   // GBK_TO_UNICODE[9557] := 16#6B54;
   // GBK_TO_UNICODE[9558] := 16#9A5C;
   // GBK_TO_UNICODE[9559] := 16#6B55;
   // GBK_TO_UNICODE[9560] := 16#9A5D;
   // GBK_TO_UNICODE[9561] := 16#6B56;
   // GBK_TO_UNICODE[9562] := 16#9A5E;
   // GBK_TO_UNICODE[9563] := 16#6B57;
   // GBK_TO_UNICODE[9564] := 16#9A5F;
   // GBK_TO_UNICODE[9565] := 16#6B58;
   // GBK_TO_UNICODE[9566] := 16#9A60;
   // GBK_TO_UNICODE[9567] := 16#6B5A;
   // GBK_TO_UNICODE[9568] := 16#9A61;
   // GBK_TO_UNICODE[9569] := 16#6B5B;
   // GBK_TO_UNICODE[9570] := 16#9A62;
   // GBK_TO_UNICODE[9571] := 16#6B5C;
   // GBK_TO_UNICODE[9572] := 16#9A63;
   // GBK_TO_UNICODE[9573] := 16#6B5D;
   // GBK_TO_UNICODE[9574] := 16#9A64;
   // GBK_TO_UNICODE[9575] := 16#6B5E;
   // GBK_TO_UNICODE[9576] := 16#9A65;
   // GBK_TO_UNICODE[9577] := 16#6B5F;
   // GBK_TO_UNICODE[9578] := 16#9A66;
   // GBK_TO_UNICODE[9579] := 16#6B60;
   // GBK_TO_UNICODE[9580] := 16#9A67;
   // GBK_TO_UNICODE[9581] := 16#6B61;
   // GBK_TO_UNICODE[9582] := 16#9A68;
   // GBK_TO_UNICODE[9583] := 16#6B68;
   // GBK_TO_UNICODE[9584] := 16#9A69;
   // GBK_TO_UNICODE[9585] := 16#6B69;
   // GBK_TO_UNICODE[9586] := 16#9A6A;
   // GBK_TO_UNICODE[9587] := 16#6B6B;
   // GBK_TO_UNICODE[9588] := 16#9A6B;
   // GBK_TO_UNICODE[9589] := 16#6B6C;
   // GBK_TO_UNICODE[9590] := 16#9A6C;
   // GBK_TO_UNICODE[9591] := 16#6B6D;
   // GBK_TO_UNICODE[9592] := 16#9A6D;
   // GBK_TO_UNICODE[9593] := 16#6B6E;
   // GBK_TO_UNICODE[9594] := 16#9A6E;
   // GBK_TO_UNICODE[9595] := 16#6B6F;
   // GBK_TO_UNICODE[9596] := 16#9A6F;
   // GBK_TO_UNICODE[9597] := 16#6B70;
   // GBK_TO_UNICODE[9598] := 16#9A70;
   // GBK_TO_UNICODE[9599] := 16#6B71;
   // GBK_TO_UNICODE[9600] := 16#9A71;
   // GBK_TO_UNICODE[9601] := 16#6B72;
   // GBK_TO_UNICODE[9602] := 16#9A72;
   // GBK_TO_UNICODE[9603] := 16#6B73;
   // GBK_TO_UNICODE[9604] := 16#9A73;
   // GBK_TO_UNICODE[9605] := 16#6B74;
   // GBK_TO_UNICODE[9606] := 16#9A74;
   // GBK_TO_UNICODE[9607] := 16#6B75;
   // GBK_TO_UNICODE[9608] := 16#9A75;
   // GBK_TO_UNICODE[9609] := 16#6B76;
   // GBK_TO_UNICODE[9610] := 16#9A76;
   // GBK_TO_UNICODE[9611] := 16#6B77;
   // GBK_TO_UNICODE[9612] := 16#9A77;
   // GBK_TO_UNICODE[9613] := 16#6B78;
   // GBK_TO_UNICODE[9614] := 16#9A78;
   // GBK_TO_UNICODE[9615] := 16#6B7A;
   // GBK_TO_UNICODE[9616] := 16#9A79;
   // GBK_TO_UNICODE[9617] := 16#6B7D;
   // GBK_TO_UNICODE[9618] := 16#9A7A;
   // GBK_TO_UNICODE[9619] := 16#6B7E;
   // GBK_TO_UNICODE[9620] := 16#9A7B;
   // GBK_TO_UNICODE[9621] := 16#6B7F;
   // GBK_TO_UNICODE[9622] := 16#9A7C;
   // GBK_TO_UNICODE[9623] := 16#6B80;
   // GBK_TO_UNICODE[9624] := 16#9A7D;
   // GBK_TO_UNICODE[9625] := 16#6B85;
   // GBK_TO_UNICODE[9626] := 16#9A7E;
   // GBK_TO_UNICODE[9627] := 16#6B88;
   // GBK_TO_UNICODE[9628] := 16#9A80;
   // GBK_TO_UNICODE[9629] := 16#6B8C;
   // GBK_TO_UNICODE[9630] := 16#9A81;
   // GBK_TO_UNICODE[9631] := 16#6B8E;
   // GBK_TO_UNICODE[9632] := 16#9A82;
   // GBK_TO_UNICODE[9633] := 16#6B8F;
   // GBK_TO_UNICODE[9634] := 16#9A83;
   // GBK_TO_UNICODE[9635] := 16#6B90;
   // GBK_TO_UNICODE[9636] := 16#9A84;
   // GBK_TO_UNICODE[9637] := 16#6B91;
   // GBK_TO_UNICODE[9638] := 16#9A85;
   // GBK_TO_UNICODE[9639] := 16#6B94;
   // GBK_TO_UNICODE[9640] := 16#9A86;
   // GBK_TO_UNICODE[9641] := 16#6B95;
   // GBK_TO_UNICODE[9642] := 16#9A87;
   // GBK_TO_UNICODE[9643] := 16#6B97;
   // GBK_TO_UNICODE[9644] := 16#9A88;
   // GBK_TO_UNICODE[9645] := 16#6B98;
   // GBK_TO_UNICODE[9646] := 16#9A89;
   // GBK_TO_UNICODE[9647] := 16#6B99;
   // GBK_TO_UNICODE[9648] := 16#9A8A;
   // GBK_TO_UNICODE[9649] := 16#6B9C;
   // GBK_TO_UNICODE[9650] := 16#9A8B;
   // GBK_TO_UNICODE[9651] := 16#6B9D;
   // GBK_TO_UNICODE[9652] := 16#9A8C;
   // GBK_TO_UNICODE[9653] := 16#6B9E;
   // GBK_TO_UNICODE[9654] := 16#9A8D;
   // GBK_TO_UNICODE[9655] := 16#6B9F;
   // GBK_TO_UNICODE[9656] := 16#9A8E;
   // GBK_TO_UNICODE[9657] := 16#6BA0;
   // GBK_TO_UNICODE[9658] := 16#9A8F;
   // GBK_TO_UNICODE[9659] := 16#6BA2;
   // GBK_TO_UNICODE[9660] := 16#9A90;
   // GBK_TO_UNICODE[9661] := 16#6BA3;
   // GBK_TO_UNICODE[9662] := 16#9A91;
   // GBK_TO_UNICODE[9663] := 16#6BA4;
   // GBK_TO_UNICODE[9664] := 16#9A92;
   // GBK_TO_UNICODE[9665] := 16#6BA5;
   // GBK_TO_UNICODE[9666] := 16#9A93;
   // GBK_TO_UNICODE[9667] := 16#6BA6;
   // GBK_TO_UNICODE[9668] := 16#9A94;
   // GBK_TO_UNICODE[9669] := 16#6BA7;
   // GBK_TO_UNICODE[9670] := 16#9A95;
   // GBK_TO_UNICODE[9671] := 16#6BA8;
   // GBK_TO_UNICODE[9672] := 16#9A96;
   // GBK_TO_UNICODE[9673] := 16#6BA9;
   // GBK_TO_UNICODE[9674] := 16#9A97;
   // GBK_TO_UNICODE[9675] := 16#6BAB;
   // GBK_TO_UNICODE[9676] := 16#9A98;
   // GBK_TO_UNICODE[9677] := 16#6BAC;
   // GBK_TO_UNICODE[9678] := 16#9A99;
   // GBK_TO_UNICODE[9679] := 16#6BAD;
   // GBK_TO_UNICODE[9680] := 16#9A9A;
   // GBK_TO_UNICODE[9681] := 16#6BAE;
   // GBK_TO_UNICODE[9682] := 16#9A9B;
   // GBK_TO_UNICODE[9683] := 16#6BAF;
   // GBK_TO_UNICODE[9684] := 16#9A9C;
   // GBK_TO_UNICODE[9685] := 16#6BB0;
   // GBK_TO_UNICODE[9686] := 16#9A9D;
   // GBK_TO_UNICODE[9687] := 16#6BB1;
   // GBK_TO_UNICODE[9688] := 16#9A9E;
   // GBK_TO_UNICODE[9689] := 16#6BB2;
   // GBK_TO_UNICODE[9690] := 16#9A9F;
   // GBK_TO_UNICODE[9691] := 16#6BB6;
   // GBK_TO_UNICODE[9692] := 16#9AA0;
   // GBK_TO_UNICODE[9693] := 16#6BB8;
   // GBK_TO_UNICODE[9694] := 16#9AA1;
   // GBK_TO_UNICODE[9695] := 16#6BB9;
   // GBK_TO_UNICODE[9696] := 16#9AA2;
   // GBK_TO_UNICODE[9697] := 16#6BBA;
   // GBK_TO_UNICODE[9698] := 16#9AA3;
   // GBK_TO_UNICODE[9699] := 16#6BBB;
   // GBK_TO_UNICODE[9700] := 16#9AA4;
   // GBK_TO_UNICODE[9701] := 16#6BBC;
   // GBK_TO_UNICODE[9702] := 16#9AA5;
   // GBK_TO_UNICODE[9703] := 16#6BBD;
   // GBK_TO_UNICODE[9704] := 16#9AA6;
   // GBK_TO_UNICODE[9705] := 16#6BBE;
   // GBK_TO_UNICODE[9706] := 16#9AA7;
   // GBK_TO_UNICODE[9707] := 16#6BC0;
   // GBK_TO_UNICODE[9708] := 16#9AA8;
   // GBK_TO_UNICODE[9709] := 16#6BC3;
   // GBK_TO_UNICODE[9710] := 16#9AA9;
   // GBK_TO_UNICODE[9711] := 16#6BC4;
   // GBK_TO_UNICODE[9712] := 16#9AAA;
   // GBK_TO_UNICODE[9713] := 16#6BC6;
   // GBK_TO_UNICODE[9714] := 16#9AAB;
   // GBK_TO_UNICODE[9715] := 16#6BC7;
   // GBK_TO_UNICODE[9716] := 16#9AAC;
   // GBK_TO_UNICODE[9717] := 16#6BC8;
   // GBK_TO_UNICODE[9718] := 16#9AAD;
   // GBK_TO_UNICODE[9719] := 16#6BC9;
   // GBK_TO_UNICODE[9720] := 16#9AAE;
   // GBK_TO_UNICODE[9721] := 16#6BCA;
   // GBK_TO_UNICODE[9722] := 16#9AAF;
   // GBK_TO_UNICODE[9723] := 16#6BCC;
   // GBK_TO_UNICODE[9724] := 16#9AB0;
   // GBK_TO_UNICODE[9725] := 16#6BCE;
   // GBK_TO_UNICODE[9726] := 16#9AB1;
   // GBK_TO_UNICODE[9727] := 16#6BD0;
   // GBK_TO_UNICODE[9728] := 16#9AB2;
   // GBK_TO_UNICODE[9729] := 16#6BD1;
   // GBK_TO_UNICODE[9730] := 16#9AB3;
   // GBK_TO_UNICODE[9731] := 16#6BD8;
   // GBK_TO_UNICODE[9732] := 16#9AB4;
   // GBK_TO_UNICODE[9733] := 16#6BDA;
   // GBK_TO_UNICODE[9734] := 16#9AB5;
   // GBK_TO_UNICODE[9735] := 16#6BDC;
   // GBK_TO_UNICODE[9736] := 16#9AB6;
   // GBK_TO_UNICODE[9737] := 16#6BDD;
   // GBK_TO_UNICODE[9738] := 16#9AB7;
   // GBK_TO_UNICODE[9739] := 16#6BDE;
   // GBK_TO_UNICODE[9740] := 16#9AB8;
   // GBK_TO_UNICODE[9741] := 16#6BDF;
   // GBK_TO_UNICODE[9742] := 16#9AB9;
   // GBK_TO_UNICODE[9743] := 16#6BE0;
   // GBK_TO_UNICODE[9744] := 16#9ABA;
   // GBK_TO_UNICODE[9745] := 16#6BE2;
   // GBK_TO_UNICODE[9746] := 16#9ABB;
   // GBK_TO_UNICODE[9747] := 16#6BE3;
   // GBK_TO_UNICODE[9748] := 16#9ABC;
   // GBK_TO_UNICODE[9749] := 16#6BE4;
   // GBK_TO_UNICODE[9750] := 16#9ABD;
   // GBK_TO_UNICODE[9751] := 16#6BE5;
   // GBK_TO_UNICODE[9752] := 16#9ABE;
   // GBK_TO_UNICODE[9753] := 16#6BE6;
   // GBK_TO_UNICODE[9754] := 16#9ABF;
   // GBK_TO_UNICODE[9755] := 16#6BE7;
   // GBK_TO_UNICODE[9756] := 16#9AC0;
   // GBK_TO_UNICODE[9757] := 16#6BE8;
   // GBK_TO_UNICODE[9758] := 16#9AC1;
   // GBK_TO_UNICODE[9759] := 16#6BE9;
   // GBK_TO_UNICODE[9760] := 16#9AC2;
   // GBK_TO_UNICODE[9761] := 16#6BEC;
   // GBK_TO_UNICODE[9762] := 16#9AC3;
   // GBK_TO_UNICODE[9763] := 16#6BED;
   // GBK_TO_UNICODE[9764] := 16#9AC4;
   // GBK_TO_UNICODE[9765] := 16#6BEE;
   // GBK_TO_UNICODE[9766] := 16#9AC5;
   // GBK_TO_UNICODE[9767] := 16#6BF0;
   // GBK_TO_UNICODE[9768] := 16#9AC6;
   // GBK_TO_UNICODE[9769] := 16#6BF1;
   // GBK_TO_UNICODE[9770] := 16#9AC7;
   // GBK_TO_UNICODE[9771] := 16#6BF2;
   // GBK_TO_UNICODE[9772] := 16#9AC8;
   // GBK_TO_UNICODE[9773] := 16#6BF4;
   // GBK_TO_UNICODE[9774] := 16#9AC9;
   // GBK_TO_UNICODE[9775] := 16#6BF6;
   // GBK_TO_UNICODE[9776] := 16#9ACA;
   // GBK_TO_UNICODE[9777] := 16#6BF7;
   // GBK_TO_UNICODE[9778] := 16#9ACB;
   // GBK_TO_UNICODE[9779] := 16#6BF8;
   // GBK_TO_UNICODE[9780] := 16#9ACC;
   // GBK_TO_UNICODE[9781] := 16#6BFA;
   // GBK_TO_UNICODE[9782] := 16#9ACD;
   // GBK_TO_UNICODE[9783] := 16#6BFB;
   // GBK_TO_UNICODE[9784] := 16#9ACE;
   // GBK_TO_UNICODE[9785] := 16#6BFC;
   // GBK_TO_UNICODE[9786] := 16#9ACF;
   // GBK_TO_UNICODE[9787] := 16#6BFE;
   // GBK_TO_UNICODE[9788] := 16#9AD0;
   // GBK_TO_UNICODE[9789] := 16#6BFF;
   // GBK_TO_UNICODE[9790] := 16#9AD1;
   // GBK_TO_UNICODE[9791] := 16#6C00;
   // GBK_TO_UNICODE[9792] := 16#9AD2;
   // GBK_TO_UNICODE[9793] := 16#6C01;
   // GBK_TO_UNICODE[9794] := 16#9AD3;
   // GBK_TO_UNICODE[9795] := 16#6C02;
   // GBK_TO_UNICODE[9796] := 16#9AD4;
   // GBK_TO_UNICODE[9797] := 16#6C03;
   // GBK_TO_UNICODE[9798] := 16#9AD5;
   // GBK_TO_UNICODE[9799] := 16#6C04;
   // GBK_TO_UNICODE[9800] := 16#9AD6;
   // GBK_TO_UNICODE[9801] := 16#6C08;
   // GBK_TO_UNICODE[9802] := 16#9AD7;
   // GBK_TO_UNICODE[9803] := 16#6C09;
   // GBK_TO_UNICODE[9804] := 16#9AD8;
   // GBK_TO_UNICODE[9805] := 16#6C0A;
   // GBK_TO_UNICODE[9806] := 16#9AD9;
   // GBK_TO_UNICODE[9807] := 16#6C0B;
   // GBK_TO_UNICODE[9808] := 16#9ADA;
   // GBK_TO_UNICODE[9809] := 16#6C0C;
   // GBK_TO_UNICODE[9810] := 16#9ADB;
   // GBK_TO_UNICODE[9811] := 16#6C0E;
   // GBK_TO_UNICODE[9812] := 16#9ADC;
   // GBK_TO_UNICODE[9813] := 16#6C12;
   // GBK_TO_UNICODE[9814] := 16#9ADD;
   // GBK_TO_UNICODE[9815] := 16#6C17;
   // GBK_TO_UNICODE[9816] := 16#9ADE;
   // GBK_TO_UNICODE[9817] := 16#6C1C;
   // GBK_TO_UNICODE[9818] := 16#9ADF;
   // GBK_TO_UNICODE[9819] := 16#6C1D;
   // GBK_TO_UNICODE[9820] := 16#9AE0;
   // GBK_TO_UNICODE[9821] := 16#6C1E;
   // GBK_TO_UNICODE[9822] := 16#9AE1;
   // GBK_TO_UNICODE[9823] := 16#6C20;
   // GBK_TO_UNICODE[9824] := 16#9AE2;
   // GBK_TO_UNICODE[9825] := 16#6C23;
   // GBK_TO_UNICODE[9826] := 16#9AE3;
   // GBK_TO_UNICODE[9827] := 16#6C25;
   // GBK_TO_UNICODE[9828] := 16#9AE4;
   // GBK_TO_UNICODE[9829] := 16#6C2B;
   // GBK_TO_UNICODE[9830] := 16#9AE5;
   // GBK_TO_UNICODE[9831] := 16#6C2C;
   // GBK_TO_UNICODE[9832] := 16#9AE6;
   // GBK_TO_UNICODE[9833] := 16#6C2D;
   // GBK_TO_UNICODE[9834] := 16#9AE7;
   // GBK_TO_UNICODE[9835] := 16#6C31;
   // GBK_TO_UNICODE[9836] := 16#9AE8;
   // GBK_TO_UNICODE[9837] := 16#6C33;
   // GBK_TO_UNICODE[9838] := 16#9AE9;
   // GBK_TO_UNICODE[9839] := 16#6C36;
   // GBK_TO_UNICODE[9840] := 16#9AEA;
   // GBK_TO_UNICODE[9841] := 16#6C37;
   // GBK_TO_UNICODE[9842] := 16#9AEB;
   // GBK_TO_UNICODE[9843] := 16#6C39;
   // GBK_TO_UNICODE[9844] := 16#9AEC;
   // GBK_TO_UNICODE[9845] := 16#6C3A;
   // GBK_TO_UNICODE[9846] := 16#9AED;
   // GBK_TO_UNICODE[9847] := 16#6C3B;
   // GBK_TO_UNICODE[9848] := 16#9AEE;
   // GBK_TO_UNICODE[9849] := 16#6C3C;
   // GBK_TO_UNICODE[9850] := 16#9AEF;
   // GBK_TO_UNICODE[9851] := 16#6C3E;
   // GBK_TO_UNICODE[9852] := 16#9AF0;
   // GBK_TO_UNICODE[9853] := 16#6C3F;
   // GBK_TO_UNICODE[9854] := 16#9AF1;
   // GBK_TO_UNICODE[9855] := 16#6C43;
   // GBK_TO_UNICODE[9856] := 16#9AF2;
   // GBK_TO_UNICODE[9857] := 16#6C44;
   // GBK_TO_UNICODE[9858] := 16#9AF3;
   // GBK_TO_UNICODE[9859] := 16#6C45;
   // GBK_TO_UNICODE[9860] := 16#9AF4;
   // GBK_TO_UNICODE[9861] := 16#6C48;
   // GBK_TO_UNICODE[9862] := 16#9AF5;
   // GBK_TO_UNICODE[9863] := 16#6C4B;
   // GBK_TO_UNICODE[9864] := 16#9AF6;
   // GBK_TO_UNICODE[9865] := 16#6C4C;
   // GBK_TO_UNICODE[9866] := 16#9AF7;
   // GBK_TO_UNICODE[9867] := 16#6C4D;
   // GBK_TO_UNICODE[9868] := 16#9AF8;
   // GBK_TO_UNICODE[9869] := 16#6C4E;
   // GBK_TO_UNICODE[9870] := 16#9AF9;
   // GBK_TO_UNICODE[9871] := 16#6C4F;
   // GBK_TO_UNICODE[9872] := 16#9AFA;
   // GBK_TO_UNICODE[9873] := 16#6C51;
   // GBK_TO_UNICODE[9874] := 16#9AFB;
   // GBK_TO_UNICODE[9875] := 16#6C52;
   // GBK_TO_UNICODE[9876] := 16#9AFC;
   // GBK_TO_UNICODE[9877] := 16#6C53;
   // GBK_TO_UNICODE[9878] := 16#9AFD;
   // GBK_TO_UNICODE[9879] := 16#6C56;
   // GBK_TO_UNICODE[9880] := 16#9AFE;
   // GBK_TO_UNICODE[9881] := 16#6C58;
   // GBK_TO_UNICODE[9882] := 16#9B40;
   // GBK_TO_UNICODE[9883] := 16#6C59;
   // GBK_TO_UNICODE[9884] := 16#9B41;
   // GBK_TO_UNICODE[9885] := 16#6C5A;
   // GBK_TO_UNICODE[9886] := 16#9B42;
   // GBK_TO_UNICODE[9887] := 16#6C62;
   // GBK_TO_UNICODE[9888] := 16#9B43;
   // GBK_TO_UNICODE[9889] := 16#6C63;
   // GBK_TO_UNICODE[9890] := 16#9B44;
   // GBK_TO_UNICODE[9891] := 16#6C65;
   // GBK_TO_UNICODE[9892] := 16#9B45;
   // GBK_TO_UNICODE[9893] := 16#6C66;
   // GBK_TO_UNICODE[9894] := 16#9B46;
   // GBK_TO_UNICODE[9895] := 16#6C67;
   // GBK_TO_UNICODE[9896] := 16#9B47;
   // GBK_TO_UNICODE[9897] := 16#6C6B;
   // GBK_TO_UNICODE[9898] := 16#9B48;
   // GBK_TO_UNICODE[9899] := 16#6C6C;
   // GBK_TO_UNICODE[9900] := 16#9B49;
   // GBK_TO_UNICODE[9901] := 16#6C6D;
   // GBK_TO_UNICODE[9902] := 16#9B4A;
   // GBK_TO_UNICODE[9903] := 16#6C6E;
   // GBK_TO_UNICODE[9904] := 16#9B4B;
   // GBK_TO_UNICODE[9905] := 16#6C6F;
   // GBK_TO_UNICODE[9906] := 16#9B4C;
   // GBK_TO_UNICODE[9907] := 16#6C71;
   // GBK_TO_UNICODE[9908] := 16#9B4D;
   // GBK_TO_UNICODE[9909] := 16#6C73;
   // GBK_TO_UNICODE[9910] := 16#9B4E;
   // GBK_TO_UNICODE[9911] := 16#6C75;
   // GBK_TO_UNICODE[9912] := 16#9B4F;
   // GBK_TO_UNICODE[9913] := 16#6C77;
   // GBK_TO_UNICODE[9914] := 16#9B50;
   // GBK_TO_UNICODE[9915] := 16#6C78;
   // GBK_TO_UNICODE[9916] := 16#9B51;
   // GBK_TO_UNICODE[9917] := 16#6C7A;
   // GBK_TO_UNICODE[9918] := 16#9B52;
   // GBK_TO_UNICODE[9919] := 16#6C7B;
   // GBK_TO_UNICODE[9920] := 16#9B53;
   // GBK_TO_UNICODE[9921] := 16#6C7C;
   // GBK_TO_UNICODE[9922] := 16#9B54;
   // GBK_TO_UNICODE[9923] := 16#6C7F;
   // GBK_TO_UNICODE[9924] := 16#9B55;
   // GBK_TO_UNICODE[9925] := 16#6C80;
   // GBK_TO_UNICODE[9926] := 16#9B56;
   // GBK_TO_UNICODE[9927] := 16#6C84;
   // GBK_TO_UNICODE[9928] := 16#9B57;
   // GBK_TO_UNICODE[9929] := 16#6C87;
   // GBK_TO_UNICODE[9930] := 16#9B58;
   // GBK_TO_UNICODE[9931] := 16#6C8A;
   // GBK_TO_UNICODE[9932] := 16#9B59;
   // GBK_TO_UNICODE[9933] := 16#6C8B;
   // GBK_TO_UNICODE[9934] := 16#9B5A;
   // GBK_TO_UNICODE[9935] := 16#6C8D;
   // GBK_TO_UNICODE[9936] := 16#9B5B;
   // GBK_TO_UNICODE[9937] := 16#6C8E;
   // GBK_TO_UNICODE[9938] := 16#9B5C;
   // GBK_TO_UNICODE[9939] := 16#6C91;
   // GBK_TO_UNICODE[9940] := 16#9B5D;
   // GBK_TO_UNICODE[9941] := 16#6C92;
   // GBK_TO_UNICODE[9942] := 16#9B5E;
   // GBK_TO_UNICODE[9943] := 16#6C95;
   // GBK_TO_UNICODE[9944] := 16#9B5F;
   // GBK_TO_UNICODE[9945] := 16#6C96;
   // GBK_TO_UNICODE[9946] := 16#9B60;
   // GBK_TO_UNICODE[9947] := 16#6C97;
   // GBK_TO_UNICODE[9948] := 16#9B61;
   // GBK_TO_UNICODE[9949] := 16#6C98;
   // GBK_TO_UNICODE[9950] := 16#9B62;
   // GBK_TO_UNICODE[9951] := 16#6C9A;
   // GBK_TO_UNICODE[9952] := 16#9B63;
   // GBK_TO_UNICODE[9953] := 16#6C9C;
   // GBK_TO_UNICODE[9954] := 16#9B64;
   // GBK_TO_UNICODE[9955] := 16#6C9D;
   // GBK_TO_UNICODE[9956] := 16#9B65;
   // GBK_TO_UNICODE[9957] := 16#6C9E;
   // GBK_TO_UNICODE[9958] := 16#9B66;
   // GBK_TO_UNICODE[9959] := 16#6CA0;
   // GBK_TO_UNICODE[9960] := 16#9B67;
   // GBK_TO_UNICODE[9961] := 16#6CA2;
   // GBK_TO_UNICODE[9962] := 16#9B68;
   // GBK_TO_UNICODE[9963] := 16#6CA8;
   // GBK_TO_UNICODE[9964] := 16#9B69;
   // GBK_TO_UNICODE[9965] := 16#6CAC;
   // GBK_TO_UNICODE[9966] := 16#9B6A;
   // GBK_TO_UNICODE[9967] := 16#6CAF;
   // GBK_TO_UNICODE[9968] := 16#9B6B;
   // GBK_TO_UNICODE[9969] := 16#6CB0;
   // GBK_TO_UNICODE[9970] := 16#9B6C;
   // GBK_TO_UNICODE[9971] := 16#6CB4;
   // GBK_TO_UNICODE[9972] := 16#9B6D;
   // GBK_TO_UNICODE[9973] := 16#6CB5;
   // GBK_TO_UNICODE[9974] := 16#9B6E;
   // GBK_TO_UNICODE[9975] := 16#6CB6;
   // GBK_TO_UNICODE[9976] := 16#9B6F;
   // GBK_TO_UNICODE[9977] := 16#6CB7;
   // GBK_TO_UNICODE[9978] := 16#9B70;
   // GBK_TO_UNICODE[9979] := 16#6CBA;
   // GBK_TO_UNICODE[9980] := 16#9B71;
   // GBK_TO_UNICODE[9981] := 16#6CC0;
   // GBK_TO_UNICODE[9982] := 16#9B72;
   // GBK_TO_UNICODE[9983] := 16#6CC1;
   // GBK_TO_UNICODE[9984] := 16#9B73;
   // GBK_TO_UNICODE[9985] := 16#6CC2;
   // GBK_TO_UNICODE[9986] := 16#9B74;
   // GBK_TO_UNICODE[9987] := 16#6CC3;
   // GBK_TO_UNICODE[9988] := 16#9B75;
   // GBK_TO_UNICODE[9989] := 16#6CC6;
   // GBK_TO_UNICODE[9990] := 16#9B76;
   // GBK_TO_UNICODE[9991] := 16#6CC7;
   // GBK_TO_UNICODE[9992] := 16#9B77;
   // GBK_TO_UNICODE[9993] := 16#6CC8;
   // GBK_TO_UNICODE[9994] := 16#9B78;
   // GBK_TO_UNICODE[9995] := 16#6CCB;
   // GBK_TO_UNICODE[9996] := 16#9B79;
   // GBK_TO_UNICODE[9997] := 16#6CCD;
   // GBK_TO_UNICODE[9998] := 16#9B7A;
   // GBK_TO_UNICODE[9999] := 16#6CCE;
   // GBK_TO_UNICODE[10000] := 16#9B7B;
   // GBK_TO_UNICODE[10001] := 16#6CCF;
   // GBK_TO_UNICODE[10002] := 16#9B7C;
   // GBK_TO_UNICODE[10003] := 16#6CD1;
   // GBK_TO_UNICODE[10004] := 16#9B7D;
   // GBK_TO_UNICODE[10005] := 16#6CD2;
   // GBK_TO_UNICODE[10006] := 16#9B7E;
   // GBK_TO_UNICODE[10007] := 16#6CD8;
   // GBK_TO_UNICODE[10008] := 16#9B80;
   // GBK_TO_UNICODE[10009] := 16#6CD9;
   // GBK_TO_UNICODE[10010] := 16#9B81;
   // GBK_TO_UNICODE[10011] := 16#6CDA;
   // GBK_TO_UNICODE[10012] := 16#9B82;
   // GBK_TO_UNICODE[10013] := 16#6CDC;
   // GBK_TO_UNICODE[10014] := 16#9B83;
   // GBK_TO_UNICODE[10015] := 16#6CDD;
   // GBK_TO_UNICODE[10016] := 16#9B84;
   // GBK_TO_UNICODE[10017] := 16#6CDF;
   // GBK_TO_UNICODE[10018] := 16#9B85;
   // GBK_TO_UNICODE[10019] := 16#6CE4;
   // GBK_TO_UNICODE[10020] := 16#9B86;
   // GBK_TO_UNICODE[10021] := 16#6CE6;
   // GBK_TO_UNICODE[10022] := 16#9B87;
   // GBK_TO_UNICODE[10023] := 16#6CE7;
   // GBK_TO_UNICODE[10024] := 16#9B88;
   // GBK_TO_UNICODE[10025] := 16#6CE9;
   // GBK_TO_UNICODE[10026] := 16#9B89;
   // GBK_TO_UNICODE[10027] := 16#6CEC;
   // GBK_TO_UNICODE[10028] := 16#9B8A;
   // GBK_TO_UNICODE[10029] := 16#6CED;
   // GBK_TO_UNICODE[10030] := 16#9B8B;
   // GBK_TO_UNICODE[10031] := 16#6CF2;
   // GBK_TO_UNICODE[10032] := 16#9B8C;
   // GBK_TO_UNICODE[10033] := 16#6CF4;
   // GBK_TO_UNICODE[10034] := 16#9B8D;
   // GBK_TO_UNICODE[10035] := 16#6CF9;
   // GBK_TO_UNICODE[10036] := 16#9B8E;
   // GBK_TO_UNICODE[10037] := 16#6CFF;
   // GBK_TO_UNICODE[10038] := 16#9B8F;
   // GBK_TO_UNICODE[10039] := 16#6D00;
   // GBK_TO_UNICODE[10040] := 16#9B90;
   // GBK_TO_UNICODE[10041] := 16#6D02;
   // GBK_TO_UNICODE[10042] := 16#9B91;
   // GBK_TO_UNICODE[10043] := 16#6D03;
   // GBK_TO_UNICODE[10044] := 16#9B92;
   // GBK_TO_UNICODE[10045] := 16#6D05;
   // GBK_TO_UNICODE[10046] := 16#9B93;
   // GBK_TO_UNICODE[10047] := 16#6D06;
   // GBK_TO_UNICODE[10048] := 16#9B94;
   // GBK_TO_UNICODE[10049] := 16#6D08;
   // GBK_TO_UNICODE[10050] := 16#9B95;
   // GBK_TO_UNICODE[10051] := 16#6D09;
   // GBK_TO_UNICODE[10052] := 16#9B96;
   // GBK_TO_UNICODE[10053] := 16#6D0A;
   // GBK_TO_UNICODE[10054] := 16#9B97;
   // GBK_TO_UNICODE[10055] := 16#6D0D;
   // GBK_TO_UNICODE[10056] := 16#9B98;
   // GBK_TO_UNICODE[10057] := 16#6D0F;
   // GBK_TO_UNICODE[10058] := 16#9B99;
   // GBK_TO_UNICODE[10059] := 16#6D10;
   // GBK_TO_UNICODE[10060] := 16#9B9A;
   // GBK_TO_UNICODE[10061] := 16#6D11;
   // GBK_TO_UNICODE[10062] := 16#9B9B;
   // GBK_TO_UNICODE[10063] := 16#6D13;
   // GBK_TO_UNICODE[10064] := 16#9B9C;
   // GBK_TO_UNICODE[10065] := 16#6D14;
   // GBK_TO_UNICODE[10066] := 16#9B9D;
   // GBK_TO_UNICODE[10067] := 16#6D15;
   // GBK_TO_UNICODE[10068] := 16#9B9E;
   // GBK_TO_UNICODE[10069] := 16#6D16;
   // GBK_TO_UNICODE[10070] := 16#9B9F;
   // GBK_TO_UNICODE[10071] := 16#6D18;
   // GBK_TO_UNICODE[10072] := 16#9BA0;
   // GBK_TO_UNICODE[10073] := 16#6D1C;
   // GBK_TO_UNICODE[10074] := 16#9BA1;
   // GBK_TO_UNICODE[10075] := 16#6D1D;
   // GBK_TO_UNICODE[10076] := 16#9BA2;
   // GBK_TO_UNICODE[10077] := 16#6D1F;
   // GBK_TO_UNICODE[10078] := 16#9BA3;
   // GBK_TO_UNICODE[10079] := 16#6D20;
   // GBK_TO_UNICODE[10080] := 16#9BA4;
   // GBK_TO_UNICODE[10081] := 16#6D21;
   // GBK_TO_UNICODE[10082] := 16#9BA5;
   // GBK_TO_UNICODE[10083] := 16#6D22;
   // GBK_TO_UNICODE[10084] := 16#9BA6;
   // GBK_TO_UNICODE[10085] := 16#6D23;
   // GBK_TO_UNICODE[10086] := 16#9BA7;
   // GBK_TO_UNICODE[10087] := 16#6D24;
   // GBK_TO_UNICODE[10088] := 16#9BA8;
   // GBK_TO_UNICODE[10089] := 16#6D26;
   // GBK_TO_UNICODE[10090] := 16#9BA9;
   // GBK_TO_UNICODE[10091] := 16#6D28;
   // GBK_TO_UNICODE[10092] := 16#9BAA;
   // GBK_TO_UNICODE[10093] := 16#6D29;
   // GBK_TO_UNICODE[10094] := 16#9BAB;
   // GBK_TO_UNICODE[10095] := 16#6D2C;
   // GBK_TO_UNICODE[10096] := 16#9BAC;
   // GBK_TO_UNICODE[10097] := 16#6D2D;
   // GBK_TO_UNICODE[10098] := 16#9BAD;
   // GBK_TO_UNICODE[10099] := 16#6D2F;
   // GBK_TO_UNICODE[10100] := 16#9BAE;
   // GBK_TO_UNICODE[10101] := 16#6D30;
   // GBK_TO_UNICODE[10102] := 16#9BAF;
   // GBK_TO_UNICODE[10103] := 16#6D34;
   // GBK_TO_UNICODE[10104] := 16#9BB0;
   // GBK_TO_UNICODE[10105] := 16#6D36;
   // GBK_TO_UNICODE[10106] := 16#9BB1;
   // GBK_TO_UNICODE[10107] := 16#6D37;
   // GBK_TO_UNICODE[10108] := 16#9BB2;
   // GBK_TO_UNICODE[10109] := 16#6D38;
   // GBK_TO_UNICODE[10110] := 16#9BB3;
   // GBK_TO_UNICODE[10111] := 16#6D3A;
   // GBK_TO_UNICODE[10112] := 16#9BB4;
   // GBK_TO_UNICODE[10113] := 16#6D3F;
   // GBK_TO_UNICODE[10114] := 16#9BB5;
   // GBK_TO_UNICODE[10115] := 16#6D40;
   // GBK_TO_UNICODE[10116] := 16#9BB6;
   // GBK_TO_UNICODE[10117] := 16#6D42;
   // GBK_TO_UNICODE[10118] := 16#9BB7;
   // GBK_TO_UNICODE[10119] := 16#6D44;
   // GBK_TO_UNICODE[10120] := 16#9BB8;
   // GBK_TO_UNICODE[10121] := 16#6D49;
   // GBK_TO_UNICODE[10122] := 16#9BB9;
   // GBK_TO_UNICODE[10123] := 16#6D4C;
   // GBK_TO_UNICODE[10124] := 16#9BBA;
   // GBK_TO_UNICODE[10125] := 16#6D50;
   // GBK_TO_UNICODE[10126] := 16#9BBB;
   // GBK_TO_UNICODE[10127] := 16#6D55;
   // GBK_TO_UNICODE[10128] := 16#9BBC;
   // GBK_TO_UNICODE[10129] := 16#6D56;
   // GBK_TO_UNICODE[10130] := 16#9BBD;
   // GBK_TO_UNICODE[10131] := 16#6D57;
   // GBK_TO_UNICODE[10132] := 16#9BBE;
   // GBK_TO_UNICODE[10133] := 16#6D58;
   // GBK_TO_UNICODE[10134] := 16#9BBF;
   // GBK_TO_UNICODE[10135] := 16#6D5B;
   // GBK_TO_UNICODE[10136] := 16#9BC0;
   // GBK_TO_UNICODE[10137] := 16#6D5D;
   // GBK_TO_UNICODE[10138] := 16#9BC1;
   // GBK_TO_UNICODE[10139] := 16#6D5F;
   // GBK_TO_UNICODE[10140] := 16#9BC2;
   // GBK_TO_UNICODE[10141] := 16#6D61;
   // GBK_TO_UNICODE[10142] := 16#9BC3;
   // GBK_TO_UNICODE[10143] := 16#6D62;
   // GBK_TO_UNICODE[10144] := 16#9BC4;
   // GBK_TO_UNICODE[10145] := 16#6D64;
   // GBK_TO_UNICODE[10146] := 16#9BC5;
   // GBK_TO_UNICODE[10147] := 16#6D65;
   // GBK_TO_UNICODE[10148] := 16#9BC6;
   // GBK_TO_UNICODE[10149] := 16#6D67;
   // GBK_TO_UNICODE[10150] := 16#9BC7;
   // GBK_TO_UNICODE[10151] := 16#6D68;
   // GBK_TO_UNICODE[10152] := 16#9BC8;
   // GBK_TO_UNICODE[10153] := 16#6D6B;
   // GBK_TO_UNICODE[10154] := 16#9BC9;
   // GBK_TO_UNICODE[10155] := 16#6D6C;
   // GBK_TO_UNICODE[10156] := 16#9BCA;
   // GBK_TO_UNICODE[10157] := 16#6D6D;
   // GBK_TO_UNICODE[10158] := 16#9BCB;
   // GBK_TO_UNICODE[10159] := 16#6D70;
   // GBK_TO_UNICODE[10160] := 16#9BCC;
   // GBK_TO_UNICODE[10161] := 16#6D71;
   // GBK_TO_UNICODE[10162] := 16#9BCD;
   // GBK_TO_UNICODE[10163] := 16#6D72;
   // GBK_TO_UNICODE[10164] := 16#9BCE;
   // GBK_TO_UNICODE[10165] := 16#6D73;
   // GBK_TO_UNICODE[10166] := 16#9BCF;
   // GBK_TO_UNICODE[10167] := 16#6D75;
   // GBK_TO_UNICODE[10168] := 16#9BD0;
   // GBK_TO_UNICODE[10169] := 16#6D76;
   // GBK_TO_UNICODE[10170] := 16#9BD1;
   // GBK_TO_UNICODE[10171] := 16#6D79;
   // GBK_TO_UNICODE[10172] := 16#9BD2;
   // GBK_TO_UNICODE[10173] := 16#6D7A;
   // GBK_TO_UNICODE[10174] := 16#9BD3;
   // GBK_TO_UNICODE[10175] := 16#6D7B;
   // GBK_TO_UNICODE[10176] := 16#9BD4;
   // GBK_TO_UNICODE[10177] := 16#6D7D;
   // GBK_TO_UNICODE[10178] := 16#9BD5;
   // GBK_TO_UNICODE[10179] := 16#6D7E;
   // GBK_TO_UNICODE[10180] := 16#9BD6;
   // GBK_TO_UNICODE[10181] := 16#6D7F;
   // GBK_TO_UNICODE[10182] := 16#9BD7;
   // GBK_TO_UNICODE[10183] := 16#6D80;
   // GBK_TO_UNICODE[10184] := 16#9BD8;
   // GBK_TO_UNICODE[10185] := 16#6D81;
   // GBK_TO_UNICODE[10186] := 16#9BD9;
   // GBK_TO_UNICODE[10187] := 16#6D83;
   // GBK_TO_UNICODE[10188] := 16#9BDA;
   // GBK_TO_UNICODE[10189] := 16#6D84;
   // GBK_TO_UNICODE[10190] := 16#9BDB;
   // GBK_TO_UNICODE[10191] := 16#6D86;
   // GBK_TO_UNICODE[10192] := 16#9BDC;
   // GBK_TO_UNICODE[10193] := 16#6D87;
   // GBK_TO_UNICODE[10194] := 16#9BDD;
   // GBK_TO_UNICODE[10195] := 16#6D8A;
   // GBK_TO_UNICODE[10196] := 16#9BDE;
   // GBK_TO_UNICODE[10197] := 16#6D8B;
   // GBK_TO_UNICODE[10198] := 16#9BDF;
   // GBK_TO_UNICODE[10199] := 16#6D8D;
   // GBK_TO_UNICODE[10200] := 16#9BE0;
   // GBK_TO_UNICODE[10201] := 16#6D8F;
   // GBK_TO_UNICODE[10202] := 16#9BE1;
   // GBK_TO_UNICODE[10203] := 16#6D90;
   // GBK_TO_UNICODE[10204] := 16#9BE2;
   // GBK_TO_UNICODE[10205] := 16#6D92;
   // GBK_TO_UNICODE[10206] := 16#9BE3;
   // GBK_TO_UNICODE[10207] := 16#6D96;
   // GBK_TO_UNICODE[10208] := 16#9BE4;
   // GBK_TO_UNICODE[10209] := 16#6D97;
   // GBK_TO_UNICODE[10210] := 16#9BE5;
   // GBK_TO_UNICODE[10211] := 16#6D98;
   // GBK_TO_UNICODE[10212] := 16#9BE6;
   // GBK_TO_UNICODE[10213] := 16#6D99;
   // GBK_TO_UNICODE[10214] := 16#9BE7;
   // GBK_TO_UNICODE[10215] := 16#6D9A;
   // GBK_TO_UNICODE[10216] := 16#9BE8;
   // GBK_TO_UNICODE[10217] := 16#6D9C;
   // GBK_TO_UNICODE[10218] := 16#9BE9;
   // GBK_TO_UNICODE[10219] := 16#6DA2;
   // GBK_TO_UNICODE[10220] := 16#9BEA;
   // GBK_TO_UNICODE[10221] := 16#6DA5;
   // GBK_TO_UNICODE[10222] := 16#9BEB;
   // GBK_TO_UNICODE[10223] := 16#6DAC;
   // GBK_TO_UNICODE[10224] := 16#9BEC;
   // GBK_TO_UNICODE[10225] := 16#6DAD;
   // GBK_TO_UNICODE[10226] := 16#9BED;
   // GBK_TO_UNICODE[10227] := 16#6DB0;
   // GBK_TO_UNICODE[10228] := 16#9BEE;
   // GBK_TO_UNICODE[10229] := 16#6DB1;
   // GBK_TO_UNICODE[10230] := 16#9BEF;
   // GBK_TO_UNICODE[10231] := 16#6DB3;
   // GBK_TO_UNICODE[10232] := 16#9BF0;
   // GBK_TO_UNICODE[10233] := 16#6DB4;
   // GBK_TO_UNICODE[10234] := 16#9BF1;
   // GBK_TO_UNICODE[10235] := 16#6DB6;
   // GBK_TO_UNICODE[10236] := 16#9BF2;
   // GBK_TO_UNICODE[10237] := 16#6DB7;
   // GBK_TO_UNICODE[10238] := 16#9BF3;
   // GBK_TO_UNICODE[10239] := 16#6DB9;
   // GBK_TO_UNICODE[10240] := 16#9BF4;
   // GBK_TO_UNICODE[10241] := 16#6DBA;
   // GBK_TO_UNICODE[10242] := 16#9BF5;
   // GBK_TO_UNICODE[10243] := 16#6DBB;
   // GBK_TO_UNICODE[10244] := 16#9BF6;
   // GBK_TO_UNICODE[10245] := 16#6DBC;
   // GBK_TO_UNICODE[10246] := 16#9BF7;
   // GBK_TO_UNICODE[10247] := 16#6DBD;
   // GBK_TO_UNICODE[10248] := 16#9BF8;
   // GBK_TO_UNICODE[10249] := 16#6DBE;
   // GBK_TO_UNICODE[10250] := 16#9BF9;
   // GBK_TO_UNICODE[10251] := 16#6DC1;
   // GBK_TO_UNICODE[10252] := 16#9BFA;
   // GBK_TO_UNICODE[10253] := 16#6DC2;
   // GBK_TO_UNICODE[10254] := 16#9BFB;
   // GBK_TO_UNICODE[10255] := 16#6DC3;
   // GBK_TO_UNICODE[10256] := 16#9BFC;
   // GBK_TO_UNICODE[10257] := 16#6DC8;
   // GBK_TO_UNICODE[10258] := 16#9BFD;
   // GBK_TO_UNICODE[10259] := 16#6DC9;
   // GBK_TO_UNICODE[10260] := 16#9BFE;
   // GBK_TO_UNICODE[10261] := 16#6DCA;
   // GBK_TO_UNICODE[10262] := 16#9C40;
   // GBK_TO_UNICODE[10263] := 16#6DCD;
   // GBK_TO_UNICODE[10264] := 16#9C41;
   // GBK_TO_UNICODE[10265] := 16#6DCE;
   // GBK_TO_UNICODE[10266] := 16#9C42;
   // GBK_TO_UNICODE[10267] := 16#6DCF;
   // GBK_TO_UNICODE[10268] := 16#9C43;
   // GBK_TO_UNICODE[10269] := 16#6DD0;
   // GBK_TO_UNICODE[10270] := 16#9C44;
   // GBK_TO_UNICODE[10271] := 16#6DD2;
   // GBK_TO_UNICODE[10272] := 16#9C45;
   // GBK_TO_UNICODE[10273] := 16#6DD3;
   // GBK_TO_UNICODE[10274] := 16#9C46;
   // GBK_TO_UNICODE[10275] := 16#6DD4;
   // GBK_TO_UNICODE[10276] := 16#9C47;
   // GBK_TO_UNICODE[10277] := 16#6DD5;
   // GBK_TO_UNICODE[10278] := 16#9C48;
   // GBK_TO_UNICODE[10279] := 16#6DD7;
   // GBK_TO_UNICODE[10280] := 16#9C49;
   // GBK_TO_UNICODE[10281] := 16#6DDA;
   // GBK_TO_UNICODE[10282] := 16#9C4A;
   // GBK_TO_UNICODE[10283] := 16#6DDB;
   // GBK_TO_UNICODE[10284] := 16#9C4B;
   // GBK_TO_UNICODE[10285] := 16#6DDC;
   // GBK_TO_UNICODE[10286] := 16#9C4C;
   // GBK_TO_UNICODE[10287] := 16#6DDF;
   // GBK_TO_UNICODE[10288] := 16#9C4D;
   // GBK_TO_UNICODE[10289] := 16#6DE2;
   // GBK_TO_UNICODE[10290] := 16#9C4E;
   // GBK_TO_UNICODE[10291] := 16#6DE3;
   // GBK_TO_UNICODE[10292] := 16#9C4F;
   // GBK_TO_UNICODE[10293] := 16#6DE5;
   // GBK_TO_UNICODE[10294] := 16#9C50;
   // GBK_TO_UNICODE[10295] := 16#6DE7;
   // GBK_TO_UNICODE[10296] := 16#9C51;
   // GBK_TO_UNICODE[10297] := 16#6DE8;
   // GBK_TO_UNICODE[10298] := 16#9C52;
   // GBK_TO_UNICODE[10299] := 16#6DE9;
   // GBK_TO_UNICODE[10300] := 16#9C53;
   // GBK_TO_UNICODE[10301] := 16#6DEA;
   // GBK_TO_UNICODE[10302] := 16#9C54;
   // GBK_TO_UNICODE[10303] := 16#6DED;
   // GBK_TO_UNICODE[10304] := 16#9C55;
   // GBK_TO_UNICODE[10305] := 16#6DEF;
   // GBK_TO_UNICODE[10306] := 16#9C56;
   // GBK_TO_UNICODE[10307] := 16#6DF0;
   // GBK_TO_UNICODE[10308] := 16#9C57;
   // GBK_TO_UNICODE[10309] := 16#6DF2;
   // GBK_TO_UNICODE[10310] := 16#9C58;
   // GBK_TO_UNICODE[10311] := 16#6DF4;
   // GBK_TO_UNICODE[10312] := 16#9C59;
   // GBK_TO_UNICODE[10313] := 16#6DF5;
   // GBK_TO_UNICODE[10314] := 16#9C5A;
   // GBK_TO_UNICODE[10315] := 16#6DF6;
   // GBK_TO_UNICODE[10316] := 16#9C5B;
   // GBK_TO_UNICODE[10317] := 16#6DF8;
   // GBK_TO_UNICODE[10318] := 16#9C5C;
   // GBK_TO_UNICODE[10319] := 16#6DFA;
   // GBK_TO_UNICODE[10320] := 16#9C5D;
   // GBK_TO_UNICODE[10321] := 16#6DFD;
   // GBK_TO_UNICODE[10322] := 16#9C5E;
   // GBK_TO_UNICODE[10323] := 16#6DFE;
   // GBK_TO_UNICODE[10324] := 16#9C5F;
   // GBK_TO_UNICODE[10325] := 16#6DFF;
   // GBK_TO_UNICODE[10326] := 16#9C60;
   // GBK_TO_UNICODE[10327] := 16#6E00;
   // GBK_TO_UNICODE[10328] := 16#9C61;
   // GBK_TO_UNICODE[10329] := 16#6E01;
   // GBK_TO_UNICODE[10330] := 16#9C62;
   // GBK_TO_UNICODE[10331] := 16#6E02;
   // GBK_TO_UNICODE[10332] := 16#9C63;
   // GBK_TO_UNICODE[10333] := 16#6E03;
   // GBK_TO_UNICODE[10334] := 16#9C64;
   // GBK_TO_UNICODE[10335] := 16#6E04;
   // GBK_TO_UNICODE[10336] := 16#9C65;
   // GBK_TO_UNICODE[10337] := 16#6E06;
   // GBK_TO_UNICODE[10338] := 16#9C66;
   // GBK_TO_UNICODE[10339] := 16#6E07;
   // GBK_TO_UNICODE[10340] := 16#9C67;
   // GBK_TO_UNICODE[10341] := 16#6E08;
   // GBK_TO_UNICODE[10342] := 16#9C68;
   // GBK_TO_UNICODE[10343] := 16#6E09;
   // GBK_TO_UNICODE[10344] := 16#9C69;
   // GBK_TO_UNICODE[10345] := 16#6E0B;
   // GBK_TO_UNICODE[10346] := 16#9C6A;
   // GBK_TO_UNICODE[10347] := 16#6E0F;
   // GBK_TO_UNICODE[10348] := 16#9C6B;
   // GBK_TO_UNICODE[10349] := 16#6E12;
   // GBK_TO_UNICODE[10350] := 16#9C6C;
   // GBK_TO_UNICODE[10351] := 16#6E13;
   // GBK_TO_UNICODE[10352] := 16#9C6D;
   // GBK_TO_UNICODE[10353] := 16#6E15;
   // GBK_TO_UNICODE[10354] := 16#9C6E;
   // GBK_TO_UNICODE[10355] := 16#6E18;
   // GBK_TO_UNICODE[10356] := 16#9C6F;
   // GBK_TO_UNICODE[10357] := 16#6E19;
   // GBK_TO_UNICODE[10358] := 16#9C70;
   // GBK_TO_UNICODE[10359] := 16#6E1B;
   // GBK_TO_UNICODE[10360] := 16#9C71;
   // GBK_TO_UNICODE[10361] := 16#6E1C;
   // GBK_TO_UNICODE[10362] := 16#9C72;
   // GBK_TO_UNICODE[10363] := 16#6E1E;
   // GBK_TO_UNICODE[10364] := 16#9C73;
   // GBK_TO_UNICODE[10365] := 16#6E1F;
   // GBK_TO_UNICODE[10366] := 16#9C74;
   // GBK_TO_UNICODE[10367] := 16#6E22;
   // GBK_TO_UNICODE[10368] := 16#9C75;
   // GBK_TO_UNICODE[10369] := 16#6E26;
   // GBK_TO_UNICODE[10370] := 16#9C76;
   // GBK_TO_UNICODE[10371] := 16#6E27;
   // GBK_TO_UNICODE[10372] := 16#9C77;
   // GBK_TO_UNICODE[10373] := 16#6E28;
   // GBK_TO_UNICODE[10374] := 16#9C78;
   // GBK_TO_UNICODE[10375] := 16#6E2A;
   // GBK_TO_UNICODE[10376] := 16#9C79;
   // GBK_TO_UNICODE[10377] := 16#6E2C;
   // GBK_TO_UNICODE[10378] := 16#9C7A;
   // GBK_TO_UNICODE[10379] := 16#6E2E;
   // GBK_TO_UNICODE[10380] := 16#9C7B;
   // GBK_TO_UNICODE[10381] := 16#6E30;
   // GBK_TO_UNICODE[10382] := 16#9C7C;
   // GBK_TO_UNICODE[10383] := 16#6E31;
   // GBK_TO_UNICODE[10384] := 16#9C7D;
   // GBK_TO_UNICODE[10385] := 16#6E33;
   // GBK_TO_UNICODE[10386] := 16#9C7E;
   // GBK_TO_UNICODE[10387] := 16#6E35;
   // GBK_TO_UNICODE[10388] := 16#9C80;
   // GBK_TO_UNICODE[10389] := 16#6E36;
   // GBK_TO_UNICODE[10390] := 16#9C81;
   // GBK_TO_UNICODE[10391] := 16#6E37;
   // GBK_TO_UNICODE[10392] := 16#9C82;
   // GBK_TO_UNICODE[10393] := 16#6E39;
   // GBK_TO_UNICODE[10394] := 16#9C83;
   // GBK_TO_UNICODE[10395] := 16#6E3B;
   // GBK_TO_UNICODE[10396] := 16#9C84;
   // GBK_TO_UNICODE[10397] := 16#6E3C;
   // GBK_TO_UNICODE[10398] := 16#9C85;
   // GBK_TO_UNICODE[10399] := 16#6E3D;
   // GBK_TO_UNICODE[10400] := 16#9C86;
   // GBK_TO_UNICODE[10401] := 16#6E3E;
   // GBK_TO_UNICODE[10402] := 16#9C87;
   // GBK_TO_UNICODE[10403] := 16#6E3F;
   // GBK_TO_UNICODE[10404] := 16#9C88;
   // GBK_TO_UNICODE[10405] := 16#6E40;
   // GBK_TO_UNICODE[10406] := 16#9C89;
   // GBK_TO_UNICODE[10407] := 16#6E41;
   // GBK_TO_UNICODE[10408] := 16#9C8A;
   // GBK_TO_UNICODE[10409] := 16#6E42;
   // GBK_TO_UNICODE[10410] := 16#9C8B;
   // GBK_TO_UNICODE[10411] := 16#6E45;
   // GBK_TO_UNICODE[10412] := 16#9C8C;
   // GBK_TO_UNICODE[10413] := 16#6E46;
   // GBK_TO_UNICODE[10414] := 16#9C8D;
   // GBK_TO_UNICODE[10415] := 16#6E47;
   // GBK_TO_UNICODE[10416] := 16#9C8E;
   // GBK_TO_UNICODE[10417] := 16#6E48;
   // GBK_TO_UNICODE[10418] := 16#9C8F;
   // GBK_TO_UNICODE[10419] := 16#6E49;
   // GBK_TO_UNICODE[10420] := 16#9C90;
   // GBK_TO_UNICODE[10421] := 16#6E4A;
   // GBK_TO_UNICODE[10422] := 16#9C91;
   // GBK_TO_UNICODE[10423] := 16#6E4B;
   // GBK_TO_UNICODE[10424] := 16#9C92;
   // GBK_TO_UNICODE[10425] := 16#6E4C;
   // GBK_TO_UNICODE[10426] := 16#9C93;
   // GBK_TO_UNICODE[10427] := 16#6E4F;
   // GBK_TO_UNICODE[10428] := 16#9C94;
   // GBK_TO_UNICODE[10429] := 16#6E50;
   // GBK_TO_UNICODE[10430] := 16#9C95;
   // GBK_TO_UNICODE[10431] := 16#6E51;
   // GBK_TO_UNICODE[10432] := 16#9C96;
   // GBK_TO_UNICODE[10433] := 16#6E52;
   // GBK_TO_UNICODE[10434] := 16#9C97;
   // GBK_TO_UNICODE[10435] := 16#6E55;
   // GBK_TO_UNICODE[10436] := 16#9C98;
   // GBK_TO_UNICODE[10437] := 16#6E57;
   // GBK_TO_UNICODE[10438] := 16#9C99;
   // GBK_TO_UNICODE[10439] := 16#6E59;
   // GBK_TO_UNICODE[10440] := 16#9C9A;
   // GBK_TO_UNICODE[10441] := 16#6E5A;
   // GBK_TO_UNICODE[10442] := 16#9C9B;
   // GBK_TO_UNICODE[10443] := 16#6E5C;
   // GBK_TO_UNICODE[10444] := 16#9C9C;
   // GBK_TO_UNICODE[10445] := 16#6E5D;
   // GBK_TO_UNICODE[10446] := 16#9C9D;
   // GBK_TO_UNICODE[10447] := 16#6E5E;
   // GBK_TO_UNICODE[10448] := 16#9C9E;
   // GBK_TO_UNICODE[10449] := 16#6E60;
   // GBK_TO_UNICODE[10450] := 16#9C9F;
   // GBK_TO_UNICODE[10451] := 16#6E61;
   // GBK_TO_UNICODE[10452] := 16#9CA0;
   // GBK_TO_UNICODE[10453] := 16#6E62;
   // GBK_TO_UNICODE[10454] := 16#9CA1;
   // GBK_TO_UNICODE[10455] := 16#6E63;
   // GBK_TO_UNICODE[10456] := 16#9CA2;
   // GBK_TO_UNICODE[10457] := 16#6E64;
   // GBK_TO_UNICODE[10458] := 16#9CA3;
   // GBK_TO_UNICODE[10459] := 16#6E65;
   // GBK_TO_UNICODE[10460] := 16#9CA4;
   // GBK_TO_UNICODE[10461] := 16#6E66;
   // GBK_TO_UNICODE[10462] := 16#9CA5;
   // GBK_TO_UNICODE[10463] := 16#6E67;
   // GBK_TO_UNICODE[10464] := 16#9CA6;
   // GBK_TO_UNICODE[10465] := 16#6E68;
   // GBK_TO_UNICODE[10466] := 16#9CA7;
   // GBK_TO_UNICODE[10467] := 16#6E69;
   // GBK_TO_UNICODE[10468] := 16#9CA8;
   // GBK_TO_UNICODE[10469] := 16#6E6A;
   // GBK_TO_UNICODE[10470] := 16#9CA9;
   // GBK_TO_UNICODE[10471] := 16#6E6C;
   // GBK_TO_UNICODE[10472] := 16#9CAA;
   // GBK_TO_UNICODE[10473] := 16#6E6D;
   // GBK_TO_UNICODE[10474] := 16#9CAB;
   // GBK_TO_UNICODE[10475] := 16#6E6F;
   // GBK_TO_UNICODE[10476] := 16#9CAC;
   // GBK_TO_UNICODE[10477] := 16#6E70;
   // GBK_TO_UNICODE[10478] := 16#9CAD;
   // GBK_TO_UNICODE[10479] := 16#6E71;
   // GBK_TO_UNICODE[10480] := 16#9CAE;
   // GBK_TO_UNICODE[10481] := 16#6E72;
   // GBK_TO_UNICODE[10482] := 16#9CAF;
   // GBK_TO_UNICODE[10483] := 16#6E73;
   // GBK_TO_UNICODE[10484] := 16#9CB0;
   // GBK_TO_UNICODE[10485] := 16#6E74;
   // GBK_TO_UNICODE[10486] := 16#9CB1;
   // GBK_TO_UNICODE[10487] := 16#6E75;
   // GBK_TO_UNICODE[10488] := 16#9CB2;
   // GBK_TO_UNICODE[10489] := 16#6E76;
   // GBK_TO_UNICODE[10490] := 16#9CB3;
   // GBK_TO_UNICODE[10491] := 16#6E77;
   // GBK_TO_UNICODE[10492] := 16#9CB4;
   // GBK_TO_UNICODE[10493] := 16#6E78;
   // GBK_TO_UNICODE[10494] := 16#9CB5;
   // GBK_TO_UNICODE[10495] := 16#6E79;
   // GBK_TO_UNICODE[10496] := 16#9CB6;
   // GBK_TO_UNICODE[10497] := 16#6E7A;
   // GBK_TO_UNICODE[10498] := 16#9CB7;
   // GBK_TO_UNICODE[10499] := 16#6E7B;
   // GBK_TO_UNICODE[10500] := 16#9CB8;
   // GBK_TO_UNICODE[10501] := 16#6E7C;
   // GBK_TO_UNICODE[10502] := 16#9CB9;
   // GBK_TO_UNICODE[10503] := 16#6E7D;
   // GBK_TO_UNICODE[10504] := 16#9CBA;
   // GBK_TO_UNICODE[10505] := 16#6E80;
   // GBK_TO_UNICODE[10506] := 16#9CBB;
   // GBK_TO_UNICODE[10507] := 16#6E81;
   // GBK_TO_UNICODE[10508] := 16#9CBC;
   // GBK_TO_UNICODE[10509] := 16#6E82;
   // GBK_TO_UNICODE[10510] := 16#9CBD;
   // GBK_TO_UNICODE[10511] := 16#6E84;
   // GBK_TO_UNICODE[10512] := 16#9CBE;
   // GBK_TO_UNICODE[10513] := 16#6E87;
   // GBK_TO_UNICODE[10514] := 16#9CBF;
   // GBK_TO_UNICODE[10515] := 16#6E88;
   // GBK_TO_UNICODE[10516] := 16#9CC0;
   // GBK_TO_UNICODE[10517] := 16#6E8A;
   // GBK_TO_UNICODE[10518] := 16#9CC1;
   // GBK_TO_UNICODE[10519] := 16#6E8B;
   // GBK_TO_UNICODE[10520] := 16#9CC2;
   // GBK_TO_UNICODE[10521] := 16#6E8C;
   // GBK_TO_UNICODE[10522] := 16#9CC3;
   // GBK_TO_UNICODE[10523] := 16#6E8D;
   // GBK_TO_UNICODE[10524] := 16#9CC4;
   // GBK_TO_UNICODE[10525] := 16#6E8E;
   // GBK_TO_UNICODE[10526] := 16#9CC5;
   // GBK_TO_UNICODE[10527] := 16#6E91;
   // GBK_TO_UNICODE[10528] := 16#9CC6;
   // GBK_TO_UNICODE[10529] := 16#6E92;
   // GBK_TO_UNICODE[10530] := 16#9CC7;
   // GBK_TO_UNICODE[10531] := 16#6E93;
   // GBK_TO_UNICODE[10532] := 16#9CC8;
   // GBK_TO_UNICODE[10533] := 16#6E94;
   // GBK_TO_UNICODE[10534] := 16#9CC9;
   // GBK_TO_UNICODE[10535] := 16#6E95;
   // GBK_TO_UNICODE[10536] := 16#9CCA;
   // GBK_TO_UNICODE[10537] := 16#6E96;
   // GBK_TO_UNICODE[10538] := 16#9CCB;
   // GBK_TO_UNICODE[10539] := 16#6E97;
   // GBK_TO_UNICODE[10540] := 16#9CCC;
   // GBK_TO_UNICODE[10541] := 16#6E99;
   // GBK_TO_UNICODE[10542] := 16#9CCD;
   // GBK_TO_UNICODE[10543] := 16#6E9A;
   // GBK_TO_UNICODE[10544] := 16#9CCE;
   // GBK_TO_UNICODE[10545] := 16#6E9B;
   // GBK_TO_UNICODE[10546] := 16#9CCF;
   // GBK_TO_UNICODE[10547] := 16#6E9D;
   // GBK_TO_UNICODE[10548] := 16#9CD0;
   // GBK_TO_UNICODE[10549] := 16#6E9E;
   // GBK_TO_UNICODE[10550] := 16#9CD1;
   // GBK_TO_UNICODE[10551] := 16#6EA0;
   // GBK_TO_UNICODE[10552] := 16#9CD2;
   // GBK_TO_UNICODE[10553] := 16#6EA1;
   // GBK_TO_UNICODE[10554] := 16#9CD3;
   // GBK_TO_UNICODE[10555] := 16#6EA3;
   // GBK_TO_UNICODE[10556] := 16#9CD4;
   // GBK_TO_UNICODE[10557] := 16#6EA4;
   // GBK_TO_UNICODE[10558] := 16#9CD5;
   // GBK_TO_UNICODE[10559] := 16#6EA6;
   // GBK_TO_UNICODE[10560] := 16#9CD6;
   // GBK_TO_UNICODE[10561] := 16#6EA8;
   // GBK_TO_UNICODE[10562] := 16#9CD7;
   // GBK_TO_UNICODE[10563] := 16#6EA9;
   // GBK_TO_UNICODE[10564] := 16#9CD8;
   // GBK_TO_UNICODE[10565] := 16#6EAB;
   // GBK_TO_UNICODE[10566] := 16#9CD9;
   // GBK_TO_UNICODE[10567] := 16#6EAC;
   // GBK_TO_UNICODE[10568] := 16#9CDA;
   // GBK_TO_UNICODE[10569] := 16#6EAD;
   // GBK_TO_UNICODE[10570] := 16#9CDB;
   // GBK_TO_UNICODE[10571] := 16#6EAE;
   // GBK_TO_UNICODE[10572] := 16#9CDC;
   // GBK_TO_UNICODE[10573] := 16#6EB0;
   // GBK_TO_UNICODE[10574] := 16#9CDD;
   // GBK_TO_UNICODE[10575] := 16#6EB3;
   // GBK_TO_UNICODE[10576] := 16#9CDE;
   // GBK_TO_UNICODE[10577] := 16#6EB5;
   // GBK_TO_UNICODE[10578] := 16#9CDF;
   // GBK_TO_UNICODE[10579] := 16#6EB8;
   // GBK_TO_UNICODE[10580] := 16#9CE0;
   // GBK_TO_UNICODE[10581] := 16#6EB9;
   // GBK_TO_UNICODE[10582] := 16#9CE1;
   // GBK_TO_UNICODE[10583] := 16#6EBC;
   // GBK_TO_UNICODE[10584] := 16#9CE2;
   // GBK_TO_UNICODE[10585] := 16#6EBE;
   // GBK_TO_UNICODE[10586] := 16#9CE3;
   // GBK_TO_UNICODE[10587] := 16#6EBF;
   // GBK_TO_UNICODE[10588] := 16#9CE4;
   // GBK_TO_UNICODE[10589] := 16#6EC0;
   // GBK_TO_UNICODE[10590] := 16#9CE5;
   // GBK_TO_UNICODE[10591] := 16#6EC3;
   // GBK_TO_UNICODE[10592] := 16#9CE6;
   // GBK_TO_UNICODE[10593] := 16#6EC4;
   // GBK_TO_UNICODE[10594] := 16#9CE7;
   // GBK_TO_UNICODE[10595] := 16#6EC5;
   // GBK_TO_UNICODE[10596] := 16#9CE8;
   // GBK_TO_UNICODE[10597] := 16#6EC6;
   // GBK_TO_UNICODE[10598] := 16#9CE9;
   // GBK_TO_UNICODE[10599] := 16#6EC8;
   // GBK_TO_UNICODE[10600] := 16#9CEA;
   // GBK_TO_UNICODE[10601] := 16#6EC9;
   // GBK_TO_UNICODE[10602] := 16#9CEB;
   // GBK_TO_UNICODE[10603] := 16#6ECA;
   // GBK_TO_UNICODE[10604] := 16#9CEC;
   // GBK_TO_UNICODE[10605] := 16#6ECC;
   // GBK_TO_UNICODE[10606] := 16#9CED;
   // GBK_TO_UNICODE[10607] := 16#6ECD;
   // GBK_TO_UNICODE[10608] := 16#9CEE;
   // GBK_TO_UNICODE[10609] := 16#6ECE;
   // GBK_TO_UNICODE[10610] := 16#9CEF;
   // GBK_TO_UNICODE[10611] := 16#6ED0;
   // GBK_TO_UNICODE[10612] := 16#9CF0;
   // GBK_TO_UNICODE[10613] := 16#6ED2;
   // GBK_TO_UNICODE[10614] := 16#9CF1;
   // GBK_TO_UNICODE[10615] := 16#6ED6;
   // GBK_TO_UNICODE[10616] := 16#9CF2;
   // GBK_TO_UNICODE[10617] := 16#6ED8;
   // GBK_TO_UNICODE[10618] := 16#9CF3;
   // GBK_TO_UNICODE[10619] := 16#6ED9;
   // GBK_TO_UNICODE[10620] := 16#9CF4;
   // GBK_TO_UNICODE[10621] := 16#6EDB;
   // GBK_TO_UNICODE[10622] := 16#9CF5;
   // GBK_TO_UNICODE[10623] := 16#6EDC;
   // GBK_TO_UNICODE[10624] := 16#9CF6;
   // GBK_TO_UNICODE[10625] := 16#6EDD;
   // GBK_TO_UNICODE[10626] := 16#9CF7;
   // GBK_TO_UNICODE[10627] := 16#6EE3;
   // GBK_TO_UNICODE[10628] := 16#9CF8;
   // GBK_TO_UNICODE[10629] := 16#6EE7;
   // GBK_TO_UNICODE[10630] := 16#9CF9;
   // GBK_TO_UNICODE[10631] := 16#6EEA;
   // GBK_TO_UNICODE[10632] := 16#9CFA;
   // GBK_TO_UNICODE[10633] := 16#6EEB;
   // GBK_TO_UNICODE[10634] := 16#9CFB;
   // GBK_TO_UNICODE[10635] := 16#6EEC;
   // GBK_TO_UNICODE[10636] := 16#9CFC;
   // GBK_TO_UNICODE[10637] := 16#6EED;
   // GBK_TO_UNICODE[10638] := 16#9CFD;
   // GBK_TO_UNICODE[10639] := 16#6EEE;
   // GBK_TO_UNICODE[10640] := 16#9CFE;
   // GBK_TO_UNICODE[10641] := 16#6EEF;
   // GBK_TO_UNICODE[10642] := 16#9D40;
   // GBK_TO_UNICODE[10643] := 16#6EF0;
   // GBK_TO_UNICODE[10644] := 16#9D41;
   // GBK_TO_UNICODE[10645] := 16#6EF1;
   // GBK_TO_UNICODE[10646] := 16#9D42;
   // GBK_TO_UNICODE[10647] := 16#6EF2;
   // GBK_TO_UNICODE[10648] := 16#9D43;
   // GBK_TO_UNICODE[10649] := 16#6EF3;
   // GBK_TO_UNICODE[10650] := 16#9D44;
   // GBK_TO_UNICODE[10651] := 16#6EF5;
   // GBK_TO_UNICODE[10652] := 16#9D45;
   // GBK_TO_UNICODE[10653] := 16#6EF6;
   // GBK_TO_UNICODE[10654] := 16#9D46;
   // GBK_TO_UNICODE[10655] := 16#6EF7;
   // GBK_TO_UNICODE[10656] := 16#9D47;
   // GBK_TO_UNICODE[10657] := 16#6EF8;
   // GBK_TO_UNICODE[10658] := 16#9D48;
   // GBK_TO_UNICODE[10659] := 16#6EFA;
   // GBK_TO_UNICODE[10660] := 16#9D49;
   // GBK_TO_UNICODE[10661] := 16#6EFB;
   // GBK_TO_UNICODE[10662] := 16#9D4A;
   // GBK_TO_UNICODE[10663] := 16#6EFC;
   // GBK_TO_UNICODE[10664] := 16#9D4B;
   // GBK_TO_UNICODE[10665] := 16#6EFD;
   // GBK_TO_UNICODE[10666] := 16#9D4C;
   // GBK_TO_UNICODE[10667] := 16#6EFE;
   // GBK_TO_UNICODE[10668] := 16#9D4D;
   // GBK_TO_UNICODE[10669] := 16#6EFF;
   // GBK_TO_UNICODE[10670] := 16#9D4E;
   // GBK_TO_UNICODE[10671] := 16#6F00;
   // GBK_TO_UNICODE[10672] := 16#9D4F;
   // GBK_TO_UNICODE[10673] := 16#6F01;
   // GBK_TO_UNICODE[10674] := 16#9D50;
   // GBK_TO_UNICODE[10675] := 16#6F03;
   // GBK_TO_UNICODE[10676] := 16#9D51;
   // GBK_TO_UNICODE[10677] := 16#6F04;
   // GBK_TO_UNICODE[10678] := 16#9D52;
   // GBK_TO_UNICODE[10679] := 16#6F05;
   // GBK_TO_UNICODE[10680] := 16#9D53;
   // GBK_TO_UNICODE[10681] := 16#6F07;
   // GBK_TO_UNICODE[10682] := 16#9D54;
   // GBK_TO_UNICODE[10683] := 16#6F08;
   // GBK_TO_UNICODE[10684] := 16#9D55;
   // GBK_TO_UNICODE[10685] := 16#6F0A;
   // GBK_TO_UNICODE[10686] := 16#9D56;
   // GBK_TO_UNICODE[10687] := 16#6F0B;
   // GBK_TO_UNICODE[10688] := 16#9D57;
   // GBK_TO_UNICODE[10689] := 16#6F0C;
   // GBK_TO_UNICODE[10690] := 16#9D58;
   // GBK_TO_UNICODE[10691] := 16#6F0D;
   // GBK_TO_UNICODE[10692] := 16#9D59;
   // GBK_TO_UNICODE[10693] := 16#6F0E;
   // GBK_TO_UNICODE[10694] := 16#9D5A;
   // GBK_TO_UNICODE[10695] := 16#6F10;
   // GBK_TO_UNICODE[10696] := 16#9D5B;
   // GBK_TO_UNICODE[10697] := 16#6F11;
   // GBK_TO_UNICODE[10698] := 16#9D5C;
   // GBK_TO_UNICODE[10699] := 16#6F12;
   // GBK_TO_UNICODE[10700] := 16#9D5D;
   // GBK_TO_UNICODE[10701] := 16#6F16;
   // GBK_TO_UNICODE[10702] := 16#9D5E;
   // GBK_TO_UNICODE[10703] := 16#6F17;
   // GBK_TO_UNICODE[10704] := 16#9D5F;
   // GBK_TO_UNICODE[10705] := 16#6F18;
   // GBK_TO_UNICODE[10706] := 16#9D60;
   // GBK_TO_UNICODE[10707] := 16#6F19;
   // GBK_TO_UNICODE[10708] := 16#9D61;
   // GBK_TO_UNICODE[10709] := 16#6F1A;
   // GBK_TO_UNICODE[10710] := 16#9D62;
   // GBK_TO_UNICODE[10711] := 16#6F1B;
   // GBK_TO_UNICODE[10712] := 16#9D63;
   // GBK_TO_UNICODE[10713] := 16#6F1C;
   // GBK_TO_UNICODE[10714] := 16#9D64;
   // GBK_TO_UNICODE[10715] := 16#6F1D;
   // GBK_TO_UNICODE[10716] := 16#9D65;
   // GBK_TO_UNICODE[10717] := 16#6F1E;
   // GBK_TO_UNICODE[10718] := 16#9D66;
   // GBK_TO_UNICODE[10719] := 16#6F1F;
   // GBK_TO_UNICODE[10720] := 16#9D67;
   // GBK_TO_UNICODE[10721] := 16#6F21;
   // GBK_TO_UNICODE[10722] := 16#9D68;
   // GBK_TO_UNICODE[10723] := 16#6F22;
   // GBK_TO_UNICODE[10724] := 16#9D69;
   // GBK_TO_UNICODE[10725] := 16#6F23;
   // GBK_TO_UNICODE[10726] := 16#9D6A;
   // GBK_TO_UNICODE[10727] := 16#6F25;
   // GBK_TO_UNICODE[10728] := 16#9D6B;
   // GBK_TO_UNICODE[10729] := 16#6F26;
   // GBK_TO_UNICODE[10730] := 16#9D6C;
   // GBK_TO_UNICODE[10731] := 16#6F27;
   // GBK_TO_UNICODE[10732] := 16#9D6D;
   // GBK_TO_UNICODE[10733] := 16#6F28;
   // GBK_TO_UNICODE[10734] := 16#9D6E;
   // GBK_TO_UNICODE[10735] := 16#6F2C;
   // GBK_TO_UNICODE[10736] := 16#9D6F;
   // GBK_TO_UNICODE[10737] := 16#6F2E;
   // GBK_TO_UNICODE[10738] := 16#9D70;
   // GBK_TO_UNICODE[10739] := 16#6F30;
   // GBK_TO_UNICODE[10740] := 16#9D71;
   // GBK_TO_UNICODE[10741] := 16#6F32;
   // GBK_TO_UNICODE[10742] := 16#9D72;
   // GBK_TO_UNICODE[10743] := 16#6F34;
   // GBK_TO_UNICODE[10744] := 16#9D73;
   // GBK_TO_UNICODE[10745] := 16#6F35;
   // GBK_TO_UNICODE[10746] := 16#9D74;
   // GBK_TO_UNICODE[10747] := 16#6F37;
   // GBK_TO_UNICODE[10748] := 16#9D75;
   // GBK_TO_UNICODE[10749] := 16#6F38;
   // GBK_TO_UNICODE[10750] := 16#9D76;
   // GBK_TO_UNICODE[10751] := 16#6F39;
   // GBK_TO_UNICODE[10752] := 16#9D77;
   // GBK_TO_UNICODE[10753] := 16#6F3A;
   // GBK_TO_UNICODE[10754] := 16#9D78;
   // GBK_TO_UNICODE[10755] := 16#6F3B;
   // GBK_TO_UNICODE[10756] := 16#9D79;
   // GBK_TO_UNICODE[10757] := 16#6F3C;
   // GBK_TO_UNICODE[10758] := 16#9D7A;
   // GBK_TO_UNICODE[10759] := 16#6F3D;
   // GBK_TO_UNICODE[10760] := 16#9D7B;
   // GBK_TO_UNICODE[10761] := 16#6F3F;
   // GBK_TO_UNICODE[10762] := 16#9D7C;
   // GBK_TO_UNICODE[10763] := 16#6F40;
   // GBK_TO_UNICODE[10764] := 16#9D7D;
   // GBK_TO_UNICODE[10765] := 16#6F41;
   // GBK_TO_UNICODE[10766] := 16#9D7E;
   // GBK_TO_UNICODE[10767] := 16#6F42;
   // GBK_TO_UNICODE[10768] := 16#9D80;
   // GBK_TO_UNICODE[10769] := 16#6F43;
   // GBK_TO_UNICODE[10770] := 16#9D81;
   // GBK_TO_UNICODE[10771] := 16#6F44;
   // GBK_TO_UNICODE[10772] := 16#9D82;
   // GBK_TO_UNICODE[10773] := 16#6F45;
   // GBK_TO_UNICODE[10774] := 16#9D83;
   // GBK_TO_UNICODE[10775] := 16#6F48;
   // GBK_TO_UNICODE[10776] := 16#9D84;
   // GBK_TO_UNICODE[10777] := 16#6F49;
   // GBK_TO_UNICODE[10778] := 16#9D85;
   // GBK_TO_UNICODE[10779] := 16#6F4A;
   // GBK_TO_UNICODE[10780] := 16#9D86;
   // GBK_TO_UNICODE[10781] := 16#6F4C;
   // GBK_TO_UNICODE[10782] := 16#9D87;
   // GBK_TO_UNICODE[10783] := 16#6F4E;
   // GBK_TO_UNICODE[10784] := 16#9D88;
   // GBK_TO_UNICODE[10785] := 16#6F4F;
   // GBK_TO_UNICODE[10786] := 16#9D89;
   // GBK_TO_UNICODE[10787] := 16#6F50;
   // GBK_TO_UNICODE[10788] := 16#9D8A;
   // GBK_TO_UNICODE[10789] := 16#6F51;
   // GBK_TO_UNICODE[10790] := 16#9D8B;
   // GBK_TO_UNICODE[10791] := 16#6F52;
   // GBK_TO_UNICODE[10792] := 16#9D8C;
   // GBK_TO_UNICODE[10793] := 16#6F53;
   // GBK_TO_UNICODE[10794] := 16#9D8D;
   // GBK_TO_UNICODE[10795] := 16#6F54;
   // GBK_TO_UNICODE[10796] := 16#9D8E;
   // GBK_TO_UNICODE[10797] := 16#6F55;
   // GBK_TO_UNICODE[10798] := 16#9D8F;
   // GBK_TO_UNICODE[10799] := 16#6F56;
   // GBK_TO_UNICODE[10800] := 16#9D90;
   // GBK_TO_UNICODE[10801] := 16#6F57;
   // GBK_TO_UNICODE[10802] := 16#9D91;
   // GBK_TO_UNICODE[10803] := 16#6F59;
   // GBK_TO_UNICODE[10804] := 16#9D92;
   // GBK_TO_UNICODE[10805] := 16#6F5A;
   // GBK_TO_UNICODE[10806] := 16#9D93;
   // GBK_TO_UNICODE[10807] := 16#6F5B;
   // GBK_TO_UNICODE[10808] := 16#9D94;
   // GBK_TO_UNICODE[10809] := 16#6F5D;
   // GBK_TO_UNICODE[10810] := 16#9D95;
   // GBK_TO_UNICODE[10811] := 16#6F5F;
   // GBK_TO_UNICODE[10812] := 16#9D96;
   // GBK_TO_UNICODE[10813] := 16#6F60;
   // GBK_TO_UNICODE[10814] := 16#9D97;
   // GBK_TO_UNICODE[10815] := 16#6F61;
   // GBK_TO_UNICODE[10816] := 16#9D98;
   // GBK_TO_UNICODE[10817] := 16#6F63;
   // GBK_TO_UNICODE[10818] := 16#9D99;
   // GBK_TO_UNICODE[10819] := 16#6F64;
   // GBK_TO_UNICODE[10820] := 16#9D9A;
   // GBK_TO_UNICODE[10821] := 16#6F65;
   // GBK_TO_UNICODE[10822] := 16#9D9B;
   // GBK_TO_UNICODE[10823] := 16#6F67;
   // GBK_TO_UNICODE[10824] := 16#9D9C;
   // GBK_TO_UNICODE[10825] := 16#6F68;
   // GBK_TO_UNICODE[10826] := 16#9D9D;
   // GBK_TO_UNICODE[10827] := 16#6F69;
   // GBK_TO_UNICODE[10828] := 16#9D9E;
   // GBK_TO_UNICODE[10829] := 16#6F6A;
   // GBK_TO_UNICODE[10830] := 16#9D9F;
   // GBK_TO_UNICODE[10831] := 16#6F6B;
   // GBK_TO_UNICODE[10832] := 16#9DA0;
   // GBK_TO_UNICODE[10833] := 16#6F6C;
   // GBK_TO_UNICODE[10834] := 16#9DA1;
   // GBK_TO_UNICODE[10835] := 16#6F6F;
   // GBK_TO_UNICODE[10836] := 16#9DA2;
   // GBK_TO_UNICODE[10837] := 16#6F70;
   // GBK_TO_UNICODE[10838] := 16#9DA3;
   // GBK_TO_UNICODE[10839] := 16#6F71;
   // GBK_TO_UNICODE[10840] := 16#9DA4;
   // GBK_TO_UNICODE[10841] := 16#6F73;
   // GBK_TO_UNICODE[10842] := 16#9DA5;
   // GBK_TO_UNICODE[10843] := 16#6F75;
   // GBK_TO_UNICODE[10844] := 16#9DA6;
   // GBK_TO_UNICODE[10845] := 16#6F76;
   // GBK_TO_UNICODE[10846] := 16#9DA7;
   // GBK_TO_UNICODE[10847] := 16#6F77;
   // GBK_TO_UNICODE[10848] := 16#9DA8;
   // GBK_TO_UNICODE[10849] := 16#6F79;
   // GBK_TO_UNICODE[10850] := 16#9DA9;
   // GBK_TO_UNICODE[10851] := 16#6F7B;
   // GBK_TO_UNICODE[10852] := 16#9DAA;
   // GBK_TO_UNICODE[10853] := 16#6F7D;
   // GBK_TO_UNICODE[10854] := 16#9DAB;
   // GBK_TO_UNICODE[10855] := 16#6F7E;
   // GBK_TO_UNICODE[10856] := 16#9DAC;
   // GBK_TO_UNICODE[10857] := 16#6F7F;
   // GBK_TO_UNICODE[10858] := 16#9DAD;
   // GBK_TO_UNICODE[10859] := 16#6F80;
   // GBK_TO_UNICODE[10860] := 16#9DAE;
   // GBK_TO_UNICODE[10861] := 16#6F81;
   // GBK_TO_UNICODE[10862] := 16#9DAF;
   // GBK_TO_UNICODE[10863] := 16#6F82;
   // GBK_TO_UNICODE[10864] := 16#9DB0;
   // GBK_TO_UNICODE[10865] := 16#6F83;
   // GBK_TO_UNICODE[10866] := 16#9DB1;
   // GBK_TO_UNICODE[10867] := 16#6F85;
   // GBK_TO_UNICODE[10868] := 16#9DB2;
   // GBK_TO_UNICODE[10869] := 16#6F86;
   // GBK_TO_UNICODE[10870] := 16#9DB3;
   // GBK_TO_UNICODE[10871] := 16#6F87;
   // GBK_TO_UNICODE[10872] := 16#9DB4;
   // GBK_TO_UNICODE[10873] := 16#6F8A;
   // GBK_TO_UNICODE[10874] := 16#9DB5;
   // GBK_TO_UNICODE[10875] := 16#6F8B;
   // GBK_TO_UNICODE[10876] := 16#9DB6;
   // GBK_TO_UNICODE[10877] := 16#6F8F;
   // GBK_TO_UNICODE[10878] := 16#9DB7;
   // GBK_TO_UNICODE[10879] := 16#6F90;
   // GBK_TO_UNICODE[10880] := 16#9DB8;
   // GBK_TO_UNICODE[10881] := 16#6F91;
   // GBK_TO_UNICODE[10882] := 16#9DB9;
   // GBK_TO_UNICODE[10883] := 16#6F92;
   // GBK_TO_UNICODE[10884] := 16#9DBA;
   // GBK_TO_UNICODE[10885] := 16#6F93;
   // GBK_TO_UNICODE[10886] := 16#9DBB;
   // GBK_TO_UNICODE[10887] := 16#6F94;
   // GBK_TO_UNICODE[10888] := 16#9DBC;
   // GBK_TO_UNICODE[10889] := 16#6F95;
   // GBK_TO_UNICODE[10890] := 16#9DBD;
   // GBK_TO_UNICODE[10891] := 16#6F96;
   // GBK_TO_UNICODE[10892] := 16#9DBE;
   // GBK_TO_UNICODE[10893] := 16#6F97;
   // GBK_TO_UNICODE[10894] := 16#9DBF;
   // GBK_TO_UNICODE[10895] := 16#6F98;
   // GBK_TO_UNICODE[10896] := 16#9DC0;
   // GBK_TO_UNICODE[10897] := 16#6F99;
   // GBK_TO_UNICODE[10898] := 16#9DC1;
   // GBK_TO_UNICODE[10899] := 16#6F9A;
   // GBK_TO_UNICODE[10900] := 16#9DC2;
   // GBK_TO_UNICODE[10901] := 16#6F9B;
   // GBK_TO_UNICODE[10902] := 16#9DC3;
   // GBK_TO_UNICODE[10903] := 16#6F9D;
   // GBK_TO_UNICODE[10904] := 16#9DC4;
   // GBK_TO_UNICODE[10905] := 16#6F9E;
   // GBK_TO_UNICODE[10906] := 16#9DC5;
   // GBK_TO_UNICODE[10907] := 16#6F9F;
   // GBK_TO_UNICODE[10908] := 16#9DC6;
   // GBK_TO_UNICODE[10909] := 16#6FA0;
   // GBK_TO_UNICODE[10910] := 16#9DC7;
   // GBK_TO_UNICODE[10911] := 16#6FA2;
   // GBK_TO_UNICODE[10912] := 16#9DC8;
   // GBK_TO_UNICODE[10913] := 16#6FA3;
   // GBK_TO_UNICODE[10914] := 16#9DC9;
   // GBK_TO_UNICODE[10915] := 16#6FA4;
   // GBK_TO_UNICODE[10916] := 16#9DCA;
   // GBK_TO_UNICODE[10917] := 16#6FA5;
   // GBK_TO_UNICODE[10918] := 16#9DCB;
   // GBK_TO_UNICODE[10919] := 16#6FA6;
   // GBK_TO_UNICODE[10920] := 16#9DCC;
   // GBK_TO_UNICODE[10921] := 16#6FA8;
   // GBK_TO_UNICODE[10922] := 16#9DCD;
   // GBK_TO_UNICODE[10923] := 16#6FA9;
   // GBK_TO_UNICODE[10924] := 16#9DCE;
   // GBK_TO_UNICODE[10925] := 16#6FAA;
   // GBK_TO_UNICODE[10926] := 16#9DCF;
   // GBK_TO_UNICODE[10927] := 16#6FAB;
   // GBK_TO_UNICODE[10928] := 16#9DD0;
   // GBK_TO_UNICODE[10929] := 16#6FAC;
   // GBK_TO_UNICODE[10930] := 16#9DD1;
   // GBK_TO_UNICODE[10931] := 16#6FAD;
   // GBK_TO_UNICODE[10932] := 16#9DD2;
   // GBK_TO_UNICODE[10933] := 16#6FAE;
   // GBK_TO_UNICODE[10934] := 16#9DD3;
   // GBK_TO_UNICODE[10935] := 16#6FAF;
   // GBK_TO_UNICODE[10936] := 16#9DD4;
   // GBK_TO_UNICODE[10937] := 16#6FB0;
   // GBK_TO_UNICODE[10938] := 16#9DD5;
   // GBK_TO_UNICODE[10939] := 16#6FB1;
   // GBK_TO_UNICODE[10940] := 16#9DD6;
   // GBK_TO_UNICODE[10941] := 16#6FB2;
   // GBK_TO_UNICODE[10942] := 16#9DD7;
   // GBK_TO_UNICODE[10943] := 16#6FB4;
   // GBK_TO_UNICODE[10944] := 16#9DD8;
   // GBK_TO_UNICODE[10945] := 16#6FB5;
   // GBK_TO_UNICODE[10946] := 16#9DD9;
   // GBK_TO_UNICODE[10947] := 16#6FB7;
   // GBK_TO_UNICODE[10948] := 16#9DDA;
   // GBK_TO_UNICODE[10949] := 16#6FB8;
   // GBK_TO_UNICODE[10950] := 16#9DDB;
   // GBK_TO_UNICODE[10951] := 16#6FBA;
   // GBK_TO_UNICODE[10952] := 16#9DDC;
   // GBK_TO_UNICODE[10953] := 16#6FBB;
   // GBK_TO_UNICODE[10954] := 16#9DDD;
   // GBK_TO_UNICODE[10955] := 16#6FBC;
   // GBK_TO_UNICODE[10956] := 16#9DDE;
   // GBK_TO_UNICODE[10957] := 16#6FBD;
   // GBK_TO_UNICODE[10958] := 16#9DDF;
   // GBK_TO_UNICODE[10959] := 16#6FBE;
   // GBK_TO_UNICODE[10960] := 16#9DE0;
   // GBK_TO_UNICODE[10961] := 16#6FBF;
   // GBK_TO_UNICODE[10962] := 16#9DE1;
   // GBK_TO_UNICODE[10963] := 16#6FC1;
   // GBK_TO_UNICODE[10964] := 16#9DE2;
   // GBK_TO_UNICODE[10965] := 16#6FC3;
   // GBK_TO_UNICODE[10966] := 16#9DE3;
   // GBK_TO_UNICODE[10967] := 16#6FC4;
   // GBK_TO_UNICODE[10968] := 16#9DE4;
   // GBK_TO_UNICODE[10969] := 16#6FC5;
   // GBK_TO_UNICODE[10970] := 16#9DE5;
   // GBK_TO_UNICODE[10971] := 16#6FC6;
   // GBK_TO_UNICODE[10972] := 16#9DE6;
   // GBK_TO_UNICODE[10973] := 16#6FC7;
   // GBK_TO_UNICODE[10974] := 16#9DE7;
   // GBK_TO_UNICODE[10975] := 16#6FC8;
   // GBK_TO_UNICODE[10976] := 16#9DE8;
   // GBK_TO_UNICODE[10977] := 16#6FCA;
   // GBK_TO_UNICODE[10978] := 16#9DE9;
   // GBK_TO_UNICODE[10979] := 16#6FCB;
   // GBK_TO_UNICODE[10980] := 16#9DEA;
   // GBK_TO_UNICODE[10981] := 16#6FCC;
   // GBK_TO_UNICODE[10982] := 16#9DEB;
   // GBK_TO_UNICODE[10983] := 16#6FCD;
   // GBK_TO_UNICODE[10984] := 16#9DEC;
   // GBK_TO_UNICODE[10985] := 16#6FCE;
   // GBK_TO_UNICODE[10986] := 16#9DED;
   // GBK_TO_UNICODE[10987] := 16#6FCF;
   // GBK_TO_UNICODE[10988] := 16#9DEE;
   // GBK_TO_UNICODE[10989] := 16#6FD0;
   // GBK_TO_UNICODE[10990] := 16#9DEF;
   // GBK_TO_UNICODE[10991] := 16#6FD3;
   // GBK_TO_UNICODE[10992] := 16#9DF0;
   // GBK_TO_UNICODE[10993] := 16#6FD4;
   // GBK_TO_UNICODE[10994] := 16#9DF1;
   // GBK_TO_UNICODE[10995] := 16#6FD5;
   // GBK_TO_UNICODE[10996] := 16#9DF2;
   // GBK_TO_UNICODE[10997] := 16#6FD6;
   // GBK_TO_UNICODE[10998] := 16#9DF3;
   // GBK_TO_UNICODE[10999] := 16#6FD7;
   // GBK_TO_UNICODE[11000] := 16#9DF4;
   // GBK_TO_UNICODE[11001] := 16#6FD8;
   // GBK_TO_UNICODE[11002] := 16#9DF5;
   // GBK_TO_UNICODE[11003] := 16#6FD9;
   // GBK_TO_UNICODE[11004] := 16#9DF6;
   // GBK_TO_UNICODE[11005] := 16#6FDA;
   // GBK_TO_UNICODE[11006] := 16#9DF7;
   // GBK_TO_UNICODE[11007] := 16#6FDB;
   // GBK_TO_UNICODE[11008] := 16#9DF8;
   // GBK_TO_UNICODE[11009] := 16#6FDC;
   // GBK_TO_UNICODE[11010] := 16#9DF9;
   // GBK_TO_UNICODE[11011] := 16#6FDD;
   // GBK_TO_UNICODE[11012] := 16#9DFA;
   // GBK_TO_UNICODE[11013] := 16#6FDF;
   // GBK_TO_UNICODE[11014] := 16#9DFB;
   // GBK_TO_UNICODE[11015] := 16#6FE2;
   // GBK_TO_UNICODE[11016] := 16#9DFC;
   // GBK_TO_UNICODE[11017] := 16#6FE3;
   // GBK_TO_UNICODE[11018] := 16#9DFD;
   // GBK_TO_UNICODE[11019] := 16#6FE4;
   // GBK_TO_UNICODE[11020] := 16#9DFE;
   // GBK_TO_UNICODE[11021] := 16#6FE5;
   // GBK_TO_UNICODE[11022] := 16#9E40;
   // GBK_TO_UNICODE[11023] := 16#6FE6;
   // GBK_TO_UNICODE[11024] := 16#9E41;
   // GBK_TO_UNICODE[11025] := 16#6FE7;
   // GBK_TO_UNICODE[11026] := 16#9E42;
   // GBK_TO_UNICODE[11027] := 16#6FE8;
   // GBK_TO_UNICODE[11028] := 16#9E43;
   // GBK_TO_UNICODE[11029] := 16#6FE9;
   // GBK_TO_UNICODE[11030] := 16#9E44;
   // GBK_TO_UNICODE[11031] := 16#6FEA;
   // GBK_TO_UNICODE[11032] := 16#9E45;
   // GBK_TO_UNICODE[11033] := 16#6FEB;
   // GBK_TO_UNICODE[11034] := 16#9E46;
   // GBK_TO_UNICODE[11035] := 16#6FEC;
   // GBK_TO_UNICODE[11036] := 16#9E47;
   // GBK_TO_UNICODE[11037] := 16#6FED;
   // GBK_TO_UNICODE[11038] := 16#9E48;
   // GBK_TO_UNICODE[11039] := 16#6FF0;
   // GBK_TO_UNICODE[11040] := 16#9E49;
   // GBK_TO_UNICODE[11041] := 16#6FF1;
   // GBK_TO_UNICODE[11042] := 16#9E4A;
   // GBK_TO_UNICODE[11043] := 16#6FF2;
   // GBK_TO_UNICODE[11044] := 16#9E4B;
   // GBK_TO_UNICODE[11045] := 16#6FF3;
   // GBK_TO_UNICODE[11046] := 16#9E4C;
   // GBK_TO_UNICODE[11047] := 16#6FF4;
   // GBK_TO_UNICODE[11048] := 16#9E4D;
   // GBK_TO_UNICODE[11049] := 16#6FF5;
   // GBK_TO_UNICODE[11050] := 16#9E4E;
   // GBK_TO_UNICODE[11051] := 16#6FF6;
   // GBK_TO_UNICODE[11052] := 16#9E4F;
   // GBK_TO_UNICODE[11053] := 16#6FF7;
   // GBK_TO_UNICODE[11054] := 16#9E50;
   // GBK_TO_UNICODE[11055] := 16#6FF8;
   // GBK_TO_UNICODE[11056] := 16#9E51;
   // GBK_TO_UNICODE[11057] := 16#6FF9;
   // GBK_TO_UNICODE[11058] := 16#9E52;
   // GBK_TO_UNICODE[11059] := 16#6FFA;
   // GBK_TO_UNICODE[11060] := 16#9E53;
   // GBK_TO_UNICODE[11061] := 16#6FFB;
   // GBK_TO_UNICODE[11062] := 16#9E54;
   // GBK_TO_UNICODE[11063] := 16#6FFC;
   // GBK_TO_UNICODE[11064] := 16#9E55;
   // GBK_TO_UNICODE[11065] := 16#6FFD;
   // GBK_TO_UNICODE[11066] := 16#9E56;
   // GBK_TO_UNICODE[11067] := 16#6FFE;
   // GBK_TO_UNICODE[11068] := 16#9E57;
   // GBK_TO_UNICODE[11069] := 16#6FFF;
   // GBK_TO_UNICODE[11070] := 16#9E58;
   // GBK_TO_UNICODE[11071] := 16#7000;
   // GBK_TO_UNICODE[11072] := 16#9E59;
   // GBK_TO_UNICODE[11073] := 16#7001;
   // GBK_TO_UNICODE[11074] := 16#9E5A;
   // GBK_TO_UNICODE[11075] := 16#7002;
   // GBK_TO_UNICODE[11076] := 16#9E5B;
   // GBK_TO_UNICODE[11077] := 16#7003;
   // GBK_TO_UNICODE[11078] := 16#9E5C;
   // GBK_TO_UNICODE[11079] := 16#7004;
   // GBK_TO_UNICODE[11080] := 16#9E5D;
   // GBK_TO_UNICODE[11081] := 16#7005;
   // GBK_TO_UNICODE[11082] := 16#9E5E;
   // GBK_TO_UNICODE[11083] := 16#7006;
   // GBK_TO_UNICODE[11084] := 16#9E5F;
   // GBK_TO_UNICODE[11085] := 16#7007;
   // GBK_TO_UNICODE[11086] := 16#9E60;
   // GBK_TO_UNICODE[11087] := 16#7008;
   // GBK_TO_UNICODE[11088] := 16#9E61;
   // GBK_TO_UNICODE[11089] := 16#7009;
   // GBK_TO_UNICODE[11090] := 16#9E62;
   // GBK_TO_UNICODE[11091] := 16#700A;
   // GBK_TO_UNICODE[11092] := 16#9E63;
   // GBK_TO_UNICODE[11093] := 16#700B;
   // GBK_TO_UNICODE[11094] := 16#9E64;
   // GBK_TO_UNICODE[11095] := 16#700C;
   // GBK_TO_UNICODE[11096] := 16#9E65;
   // GBK_TO_UNICODE[11097] := 16#700D;
   // GBK_TO_UNICODE[11098] := 16#9E66;
   // GBK_TO_UNICODE[11099] := 16#700E;
   // GBK_TO_UNICODE[11100] := 16#9E67;
   // GBK_TO_UNICODE[11101] := 16#700F;
   // GBK_TO_UNICODE[11102] := 16#9E68;
   // GBK_TO_UNICODE[11103] := 16#7010;
   // GBK_TO_UNICODE[11104] := 16#9E69;
   // GBK_TO_UNICODE[11105] := 16#7012;
   // GBK_TO_UNICODE[11106] := 16#9E6A;
   // GBK_TO_UNICODE[11107] := 16#7013;
   // GBK_TO_UNICODE[11108] := 16#9E6B;
   // GBK_TO_UNICODE[11109] := 16#7014;
   // GBK_TO_UNICODE[11110] := 16#9E6C;
   // GBK_TO_UNICODE[11111] := 16#7015;
   // GBK_TO_UNICODE[11112] := 16#9E6D;
   // GBK_TO_UNICODE[11113] := 16#7016;
   // GBK_TO_UNICODE[11114] := 16#9E6E;
   // GBK_TO_UNICODE[11115] := 16#7017;
   // GBK_TO_UNICODE[11116] := 16#9E6F;
   // GBK_TO_UNICODE[11117] := 16#7018;
   // GBK_TO_UNICODE[11118] := 16#9E70;
   // GBK_TO_UNICODE[11119] := 16#7019;
   // GBK_TO_UNICODE[11120] := 16#9E71;
   // GBK_TO_UNICODE[11121] := 16#701C;
   // GBK_TO_UNICODE[11122] := 16#9E72;
   // GBK_TO_UNICODE[11123] := 16#701D;
   // GBK_TO_UNICODE[11124] := 16#9E73;
   // GBK_TO_UNICODE[11125] := 16#701E;
   // GBK_TO_UNICODE[11126] := 16#9E74;
   // GBK_TO_UNICODE[11127] := 16#701F;
   // GBK_TO_UNICODE[11128] := 16#9E75;
   // GBK_TO_UNICODE[11129] := 16#7020;
   // GBK_TO_UNICODE[11130] := 16#9E76;
   // GBK_TO_UNICODE[11131] := 16#7021;
   // GBK_TO_UNICODE[11132] := 16#9E77;
   // GBK_TO_UNICODE[11133] := 16#7022;
   // GBK_TO_UNICODE[11134] := 16#9E78;
   // GBK_TO_UNICODE[11135] := 16#7024;
   // GBK_TO_UNICODE[11136] := 16#9E79;
   // GBK_TO_UNICODE[11137] := 16#7025;
   // GBK_TO_UNICODE[11138] := 16#9E7A;
   // GBK_TO_UNICODE[11139] := 16#7026;
   // GBK_TO_UNICODE[11140] := 16#9E7B;
   // GBK_TO_UNICODE[11141] := 16#7027;
   // GBK_TO_UNICODE[11142] := 16#9E7C;
   // GBK_TO_UNICODE[11143] := 16#7028;
   // GBK_TO_UNICODE[11144] := 16#9E7D;
   // GBK_TO_UNICODE[11145] := 16#7029;
   // GBK_TO_UNICODE[11146] := 16#9E7E;
   // GBK_TO_UNICODE[11147] := 16#702A;
   // GBK_TO_UNICODE[11148] := 16#9E80;
   // GBK_TO_UNICODE[11149] := 16#702B;
   // GBK_TO_UNICODE[11150] := 16#9E81;
   // GBK_TO_UNICODE[11151] := 16#702C;
   // GBK_TO_UNICODE[11152] := 16#9E82;
   // GBK_TO_UNICODE[11153] := 16#702D;
   // GBK_TO_UNICODE[11154] := 16#9E83;
   // GBK_TO_UNICODE[11155] := 16#702E;
   // GBK_TO_UNICODE[11156] := 16#9E84;
   // GBK_TO_UNICODE[11157] := 16#702F;
   // GBK_TO_UNICODE[11158] := 16#9E85;
   // GBK_TO_UNICODE[11159] := 16#7030;
   // GBK_TO_UNICODE[11160] := 16#9E86;
   // GBK_TO_UNICODE[11161] := 16#7031;
   // GBK_TO_UNICODE[11162] := 16#9E87;
   // GBK_TO_UNICODE[11163] := 16#7032;
   // GBK_TO_UNICODE[11164] := 16#9E88;
   // GBK_TO_UNICODE[11165] := 16#7033;
   // GBK_TO_UNICODE[11166] := 16#9E89;
   // GBK_TO_UNICODE[11167] := 16#7034;
   // GBK_TO_UNICODE[11168] := 16#9E8A;
   // GBK_TO_UNICODE[11169] := 16#7036;
   // GBK_TO_UNICODE[11170] := 16#9E8B;
   // GBK_TO_UNICODE[11171] := 16#7037;
   // GBK_TO_UNICODE[11172] := 16#9E8C;
   // GBK_TO_UNICODE[11173] := 16#7038;
   // GBK_TO_UNICODE[11174] := 16#9E8D;
   // GBK_TO_UNICODE[11175] := 16#703A;
   // GBK_TO_UNICODE[11176] := 16#9E8E;
   // GBK_TO_UNICODE[11177] := 16#703B;
   // GBK_TO_UNICODE[11178] := 16#9E8F;
   // GBK_TO_UNICODE[11179] := 16#703C;
   // GBK_TO_UNICODE[11180] := 16#9E90;
   // GBK_TO_UNICODE[11181] := 16#703D;
   // GBK_TO_UNICODE[11182] := 16#9E91;
   // GBK_TO_UNICODE[11183] := 16#703E;
   // GBK_TO_UNICODE[11184] := 16#9E92;
   // GBK_TO_UNICODE[11185] := 16#703F;
   // GBK_TO_UNICODE[11186] := 16#9E93;
   // GBK_TO_UNICODE[11187] := 16#7040;
   // GBK_TO_UNICODE[11188] := 16#9E94;
   // GBK_TO_UNICODE[11189] := 16#7041;
   // GBK_TO_UNICODE[11190] := 16#9E95;
   // GBK_TO_UNICODE[11191] := 16#7042;
   // GBK_TO_UNICODE[11192] := 16#9E96;
   // GBK_TO_UNICODE[11193] := 16#7043;
   // GBK_TO_UNICODE[11194] := 16#9E97;
   // GBK_TO_UNICODE[11195] := 16#7044;
   // GBK_TO_UNICODE[11196] := 16#9E98;
   // GBK_TO_UNICODE[11197] := 16#7045;
   // GBK_TO_UNICODE[11198] := 16#9E99;
   // GBK_TO_UNICODE[11199] := 16#7046;
   // GBK_TO_UNICODE[11200] := 16#9E9A;
   // GBK_TO_UNICODE[11201] := 16#7047;
   // GBK_TO_UNICODE[11202] := 16#9E9B;
   // GBK_TO_UNICODE[11203] := 16#7048;
   // GBK_TO_UNICODE[11204] := 16#9E9C;
   // GBK_TO_UNICODE[11205] := 16#7049;
   // GBK_TO_UNICODE[11206] := 16#9E9D;
   // GBK_TO_UNICODE[11207] := 16#704A;
   // GBK_TO_UNICODE[11208] := 16#9E9E;
   // GBK_TO_UNICODE[11209] := 16#704B;
   // GBK_TO_UNICODE[11210] := 16#9E9F;
   // GBK_TO_UNICODE[11211] := 16#704D;
   // GBK_TO_UNICODE[11212] := 16#9EA0;
   // GBK_TO_UNICODE[11213] := 16#704E;
   // GBK_TO_UNICODE[11214] := 16#9EA1;
   // GBK_TO_UNICODE[11215] := 16#7050;
   // GBK_TO_UNICODE[11216] := 16#9EA2;
   // GBK_TO_UNICODE[11217] := 16#7051;
   // GBK_TO_UNICODE[11218] := 16#9EA3;
   // GBK_TO_UNICODE[11219] := 16#7052;
   // GBK_TO_UNICODE[11220] := 16#9EA4;
   // GBK_TO_UNICODE[11221] := 16#7053;
   // GBK_TO_UNICODE[11222] := 16#9EA5;
   // GBK_TO_UNICODE[11223] := 16#7054;
   // GBK_TO_UNICODE[11224] := 16#9EA6;
   // GBK_TO_UNICODE[11225] := 16#7055;
   // GBK_TO_UNICODE[11226] := 16#9EA7;
   // GBK_TO_UNICODE[11227] := 16#7056;
   // GBK_TO_UNICODE[11228] := 16#9EA8;
   // GBK_TO_UNICODE[11229] := 16#7057;
   // GBK_TO_UNICODE[11230] := 16#9EA9;
   // GBK_TO_UNICODE[11231] := 16#7058;
   // GBK_TO_UNICODE[11232] := 16#9EAA;
   // GBK_TO_UNICODE[11233] := 16#7059;
   // GBK_TO_UNICODE[11234] := 16#9EAB;
   // GBK_TO_UNICODE[11235] := 16#705A;
   // GBK_TO_UNICODE[11236] := 16#9EAC;
   // GBK_TO_UNICODE[11237] := 16#705B;
   // GBK_TO_UNICODE[11238] := 16#9EAD;
   // GBK_TO_UNICODE[11239] := 16#705C;
   // GBK_TO_UNICODE[11240] := 16#9EAE;
   // GBK_TO_UNICODE[11241] := 16#705D;
   // GBK_TO_UNICODE[11242] := 16#9EAF;
   // GBK_TO_UNICODE[11243] := 16#705F;
   // GBK_TO_UNICODE[11244] := 16#9EB0;
   // GBK_TO_UNICODE[11245] := 16#7060;
   // GBK_TO_UNICODE[11246] := 16#9EB1;
   // GBK_TO_UNICODE[11247] := 16#7061;
   // GBK_TO_UNICODE[11248] := 16#9EB2;
   // GBK_TO_UNICODE[11249] := 16#7062;
   // GBK_TO_UNICODE[11250] := 16#9EB3;
   // GBK_TO_UNICODE[11251] := 16#7063;
   // GBK_TO_UNICODE[11252] := 16#9EB4;
   // GBK_TO_UNICODE[11253] := 16#7064;
   // GBK_TO_UNICODE[11254] := 16#9EB5;
   // GBK_TO_UNICODE[11255] := 16#7065;
   // GBK_TO_UNICODE[11256] := 16#9EB6;
   // GBK_TO_UNICODE[11257] := 16#7066;
   // GBK_TO_UNICODE[11258] := 16#9EB7;
   // GBK_TO_UNICODE[11259] := 16#7067;
   // GBK_TO_UNICODE[11260] := 16#9EB8;
   // GBK_TO_UNICODE[11261] := 16#7068;
   // GBK_TO_UNICODE[11262] := 16#9EB9;
   // GBK_TO_UNICODE[11263] := 16#7069;
   // GBK_TO_UNICODE[11264] := 16#9EBA;
   // GBK_TO_UNICODE[11265] := 16#706A;
   // GBK_TO_UNICODE[11266] := 16#9EBB;
   // GBK_TO_UNICODE[11267] := 16#706E;
   // GBK_TO_UNICODE[11268] := 16#9EBC;
   // GBK_TO_UNICODE[11269] := 16#7071;
   // GBK_TO_UNICODE[11270] := 16#9EBD;
   // GBK_TO_UNICODE[11271] := 16#7072;
   // GBK_TO_UNICODE[11272] := 16#9EBE;
   // GBK_TO_UNICODE[11273] := 16#7073;
   // GBK_TO_UNICODE[11274] := 16#9EBF;
   // GBK_TO_UNICODE[11275] := 16#7074;
   // GBK_TO_UNICODE[11276] := 16#9EC0;
   // GBK_TO_UNICODE[11277] := 16#7077;
   // GBK_TO_UNICODE[11278] := 16#9EC1;
   // GBK_TO_UNICODE[11279] := 16#7079;
   // GBK_TO_UNICODE[11280] := 16#9EC2;
   // GBK_TO_UNICODE[11281] := 16#707A;
   // GBK_TO_UNICODE[11282] := 16#9EC3;
   // GBK_TO_UNICODE[11283] := 16#707B;
   // GBK_TO_UNICODE[11284] := 16#9EC4;
   // GBK_TO_UNICODE[11285] := 16#707D;
   // GBK_TO_UNICODE[11286] := 16#9EC5;
   // GBK_TO_UNICODE[11287] := 16#7081;
   // GBK_TO_UNICODE[11288] := 16#9EC6;
   // GBK_TO_UNICODE[11289] := 16#7082;
   // GBK_TO_UNICODE[11290] := 16#9EC7;
   // GBK_TO_UNICODE[11291] := 16#7083;
   // GBK_TO_UNICODE[11292] := 16#9EC8;
   // GBK_TO_UNICODE[11293] := 16#7084;
   // GBK_TO_UNICODE[11294] := 16#9EC9;
   // GBK_TO_UNICODE[11295] := 16#7086;
   // GBK_TO_UNICODE[11296] := 16#9ECA;
   // GBK_TO_UNICODE[11297] := 16#7087;
   // GBK_TO_UNICODE[11298] := 16#9ECB;
   // GBK_TO_UNICODE[11299] := 16#7088;
   // GBK_TO_UNICODE[11300] := 16#9ECC;
   // GBK_TO_UNICODE[11301] := 16#708B;
   // GBK_TO_UNICODE[11302] := 16#9ECD;
   // GBK_TO_UNICODE[11303] := 16#708C;
   // GBK_TO_UNICODE[11304] := 16#9ECE;
   // GBK_TO_UNICODE[11305] := 16#708D;
   // GBK_TO_UNICODE[11306] := 16#9ECF;
   // GBK_TO_UNICODE[11307] := 16#708F;
   // GBK_TO_UNICODE[11308] := 16#9ED0;
   // GBK_TO_UNICODE[11309] := 16#7090;
   // GBK_TO_UNICODE[11310] := 16#9ED1;
   // GBK_TO_UNICODE[11311] := 16#7091;
   // GBK_TO_UNICODE[11312] := 16#9ED2;
   // GBK_TO_UNICODE[11313] := 16#7093;
   // GBK_TO_UNICODE[11314] := 16#9ED3;
   // GBK_TO_UNICODE[11315] := 16#7097;
   // GBK_TO_UNICODE[11316] := 16#9ED4;
   // GBK_TO_UNICODE[11317] := 16#7098;
   // GBK_TO_UNICODE[11318] := 16#9ED5;
   // GBK_TO_UNICODE[11319] := 16#709A;
   // GBK_TO_UNICODE[11320] := 16#9ED6;
   // GBK_TO_UNICODE[11321] := 16#709B;
   // GBK_TO_UNICODE[11322] := 16#9ED7;
   // GBK_TO_UNICODE[11323] := 16#709E;
   // GBK_TO_UNICODE[11324] := 16#9ED8;
   // GBK_TO_UNICODE[11325] := 16#709F;
   // GBK_TO_UNICODE[11326] := 16#9ED9;
   // GBK_TO_UNICODE[11327] := 16#70A0;
   // GBK_TO_UNICODE[11328] := 16#9EDA;
   // GBK_TO_UNICODE[11329] := 16#70A1;
   // GBK_TO_UNICODE[11330] := 16#9EDB;
   // GBK_TO_UNICODE[11331] := 16#70A2;
   // GBK_TO_UNICODE[11332] := 16#9EDC;
   // GBK_TO_UNICODE[11333] := 16#70A3;
   // GBK_TO_UNICODE[11334] := 16#9EDD;
   // GBK_TO_UNICODE[11335] := 16#70A4;
   // GBK_TO_UNICODE[11336] := 16#9EDE;
   // GBK_TO_UNICODE[11337] := 16#70A5;
   // GBK_TO_UNICODE[11338] := 16#9EDF;
   // GBK_TO_UNICODE[11339] := 16#70A6;
   // GBK_TO_UNICODE[11340] := 16#9EE0;
   // GBK_TO_UNICODE[11341] := 16#70A7;
   // GBK_TO_UNICODE[11342] := 16#9EE1;
   // GBK_TO_UNICODE[11343] := 16#70A8;
   // GBK_TO_UNICODE[11344] := 16#9EE2;
   // GBK_TO_UNICODE[11345] := 16#70A9;
   // GBK_TO_UNICODE[11346] := 16#9EE3;
   // GBK_TO_UNICODE[11347] := 16#70AA;
   // GBK_TO_UNICODE[11348] := 16#9EE4;
   // GBK_TO_UNICODE[11349] := 16#70B0;
   // GBK_TO_UNICODE[11350] := 16#9EE5;
   // GBK_TO_UNICODE[11351] := 16#70B2;
   // GBK_TO_UNICODE[11352] := 16#9EE6;
   // GBK_TO_UNICODE[11353] := 16#70B4;
   // GBK_TO_UNICODE[11354] := 16#9EE7;
   // GBK_TO_UNICODE[11355] := 16#70B5;
   // GBK_TO_UNICODE[11356] := 16#9EE8;
   // GBK_TO_UNICODE[11357] := 16#70B6;
   // GBK_TO_UNICODE[11358] := 16#9EE9;
   // GBK_TO_UNICODE[11359] := 16#70BA;
   // GBK_TO_UNICODE[11360] := 16#9EEA;
   // GBK_TO_UNICODE[11361] := 16#70BE;
   // GBK_TO_UNICODE[11362] := 16#9EEB;
   // GBK_TO_UNICODE[11363] := 16#70BF;
   // GBK_TO_UNICODE[11364] := 16#9EEC;
   // GBK_TO_UNICODE[11365] := 16#70C4;
   // GBK_TO_UNICODE[11366] := 16#9EED;
   // GBK_TO_UNICODE[11367] := 16#70C5;
   // GBK_TO_UNICODE[11368] := 16#9EEE;
   // GBK_TO_UNICODE[11369] := 16#70C6;
   // GBK_TO_UNICODE[11370] := 16#9EEF;
   // GBK_TO_UNICODE[11371] := 16#70C7;
   // GBK_TO_UNICODE[11372] := 16#9EF0;
   // GBK_TO_UNICODE[11373] := 16#70C9;
   // GBK_TO_UNICODE[11374] := 16#9EF1;
   // GBK_TO_UNICODE[11375] := 16#70CB;
   // GBK_TO_UNICODE[11376] := 16#9EF2;
   // GBK_TO_UNICODE[11377] := 16#70CC;
   // GBK_TO_UNICODE[11378] := 16#9EF3;
   // GBK_TO_UNICODE[11379] := 16#70CD;
   // GBK_TO_UNICODE[11380] := 16#9EF4;
   // GBK_TO_UNICODE[11381] := 16#70CE;
   // GBK_TO_UNICODE[11382] := 16#9EF5;
   // GBK_TO_UNICODE[11383] := 16#70CF;
   // GBK_TO_UNICODE[11384] := 16#9EF6;
   // GBK_TO_UNICODE[11385] := 16#70D0;
   // GBK_TO_UNICODE[11386] := 16#9EF7;
   // GBK_TO_UNICODE[11387] := 16#70D1;
   // GBK_TO_UNICODE[11388] := 16#9EF8;
   // GBK_TO_UNICODE[11389] := 16#70D2;
   // GBK_TO_UNICODE[11390] := 16#9EF9;
   // GBK_TO_UNICODE[11391] := 16#70D3;
   // GBK_TO_UNICODE[11392] := 16#9EFA;
   // GBK_TO_UNICODE[11393] := 16#70D4;
   // GBK_TO_UNICODE[11394] := 16#9EFB;
   // GBK_TO_UNICODE[11395] := 16#70D5;
   // GBK_TO_UNICODE[11396] := 16#9EFC;
   // GBK_TO_UNICODE[11397] := 16#70D6;
   // GBK_TO_UNICODE[11398] := 16#9EFD;
   // GBK_TO_UNICODE[11399] := 16#70D7;
   // GBK_TO_UNICODE[11400] := 16#9EFE;
   // GBK_TO_UNICODE[11401] := 16#70DA;
   // GBK_TO_UNICODE[11402] := 16#9F40;
   // GBK_TO_UNICODE[11403] := 16#70DC;
   // GBK_TO_UNICODE[11404] := 16#9F41;
   // GBK_TO_UNICODE[11405] := 16#70DD;
   // GBK_TO_UNICODE[11406] := 16#9F42;
   // GBK_TO_UNICODE[11407] := 16#70DE;
   // GBK_TO_UNICODE[11408] := 16#9F43;
   // GBK_TO_UNICODE[11409] := 16#70E0;
   // GBK_TO_UNICODE[11410] := 16#9F44;
   // GBK_TO_UNICODE[11411] := 16#70E1;
   // GBK_TO_UNICODE[11412] := 16#9F45;
   // GBK_TO_UNICODE[11413] := 16#70E2;
   // GBK_TO_UNICODE[11414] := 16#9F46;
   // GBK_TO_UNICODE[11415] := 16#70E3;
   // GBK_TO_UNICODE[11416] := 16#9F47;
   // GBK_TO_UNICODE[11417] := 16#70E5;
   // GBK_TO_UNICODE[11418] := 16#9F48;
   // GBK_TO_UNICODE[11419] := 16#70EA;
   // GBK_TO_UNICODE[11420] := 16#9F49;
   // GBK_TO_UNICODE[11421] := 16#70EE;
   // GBK_TO_UNICODE[11422] := 16#9F4A;
   // GBK_TO_UNICODE[11423] := 16#70F0;
   // GBK_TO_UNICODE[11424] := 16#9F4B;
   // GBK_TO_UNICODE[11425] := 16#70F1;
   // GBK_TO_UNICODE[11426] := 16#9F4C;
   // GBK_TO_UNICODE[11427] := 16#70F2;
   // GBK_TO_UNICODE[11428] := 16#9F4D;
   // GBK_TO_UNICODE[11429] := 16#70F3;
   // GBK_TO_UNICODE[11430] := 16#9F4E;
   // GBK_TO_UNICODE[11431] := 16#70F4;
   // GBK_TO_UNICODE[11432] := 16#9F4F;
   // GBK_TO_UNICODE[11433] := 16#70F5;
   // GBK_TO_UNICODE[11434] := 16#9F50;
   // GBK_TO_UNICODE[11435] := 16#70F6;
   // GBK_TO_UNICODE[11436] := 16#9F51;
   // GBK_TO_UNICODE[11437] := 16#70F8;
   // GBK_TO_UNICODE[11438] := 16#9F52;
   // GBK_TO_UNICODE[11439] := 16#70FA;
   // GBK_TO_UNICODE[11440] := 16#9F53;
   // GBK_TO_UNICODE[11441] := 16#70FB;
   // GBK_TO_UNICODE[11442] := 16#9F54;
   // GBK_TO_UNICODE[11443] := 16#70FC;
   // GBK_TO_UNICODE[11444] := 16#9F55;
   // GBK_TO_UNICODE[11445] := 16#70FE;
   // GBK_TO_UNICODE[11446] := 16#9F56;
   // GBK_TO_UNICODE[11447] := 16#70FF;
   // GBK_TO_UNICODE[11448] := 16#9F57;
   // GBK_TO_UNICODE[11449] := 16#7100;
   // GBK_TO_UNICODE[11450] := 16#9F58;
   // GBK_TO_UNICODE[11451] := 16#7101;
   // GBK_TO_UNICODE[11452] := 16#9F59;
   // GBK_TO_UNICODE[11453] := 16#7102;
   // GBK_TO_UNICODE[11454] := 16#9F5A;
   // GBK_TO_UNICODE[11455] := 16#7103;
   // GBK_TO_UNICODE[11456] := 16#9F5B;
   // GBK_TO_UNICODE[11457] := 16#7104;
   // GBK_TO_UNICODE[11458] := 16#9F5C;
   // GBK_TO_UNICODE[11459] := 16#7105;
   // GBK_TO_UNICODE[11460] := 16#9F5D;
   // GBK_TO_UNICODE[11461] := 16#7106;
   // GBK_TO_UNICODE[11462] := 16#9F5E;
   // GBK_TO_UNICODE[11463] := 16#7107;
   // GBK_TO_UNICODE[11464] := 16#9F5F;
   // GBK_TO_UNICODE[11465] := 16#7108;
   // GBK_TO_UNICODE[11466] := 16#9F60;
   // GBK_TO_UNICODE[11467] := 16#710B;
   // GBK_TO_UNICODE[11468] := 16#9F61;
   // GBK_TO_UNICODE[11469] := 16#710C;
   // GBK_TO_UNICODE[11470] := 16#9F62;
   // GBK_TO_UNICODE[11471] := 16#710D;
   // GBK_TO_UNICODE[11472] := 16#9F63;
   // GBK_TO_UNICODE[11473] := 16#710E;
   // GBK_TO_UNICODE[11474] := 16#9F64;
   // GBK_TO_UNICODE[11475] := 16#710F;
   // GBK_TO_UNICODE[11476] := 16#9F65;
   // GBK_TO_UNICODE[11477] := 16#7111;
   // GBK_TO_UNICODE[11478] := 16#9F66;
   // GBK_TO_UNICODE[11479] := 16#7112;
   // GBK_TO_UNICODE[11480] := 16#9F67;
   // GBK_TO_UNICODE[11481] := 16#7114;
   // GBK_TO_UNICODE[11482] := 16#9F68;
   // GBK_TO_UNICODE[11483] := 16#7117;
   // GBK_TO_UNICODE[11484] := 16#9F69;
   // GBK_TO_UNICODE[11485] := 16#711B;
   // GBK_TO_UNICODE[11486] := 16#9F6A;
   // GBK_TO_UNICODE[11487] := 16#711C;
   // GBK_TO_UNICODE[11488] := 16#9F6B;
   // GBK_TO_UNICODE[11489] := 16#711D;
   // GBK_TO_UNICODE[11490] := 16#9F6C;
   // GBK_TO_UNICODE[11491] := 16#711E;
   // GBK_TO_UNICODE[11492] := 16#9F6D;
   // GBK_TO_UNICODE[11493] := 16#711F;
   // GBK_TO_UNICODE[11494] := 16#9F6E;
   // GBK_TO_UNICODE[11495] := 16#7120;
   // GBK_TO_UNICODE[11496] := 16#9F6F;
   // GBK_TO_UNICODE[11497] := 16#7121;
   // GBK_TO_UNICODE[11498] := 16#9F70;
   // GBK_TO_UNICODE[11499] := 16#7122;
   // GBK_TO_UNICODE[11500] := 16#9F71;
   // GBK_TO_UNICODE[11501] := 16#7123;
   // GBK_TO_UNICODE[11502] := 16#9F72;
   // GBK_TO_UNICODE[11503] := 16#7124;
   // GBK_TO_UNICODE[11504] := 16#9F73;
   // GBK_TO_UNICODE[11505] := 16#7125;
   // GBK_TO_UNICODE[11506] := 16#9F74;
   // GBK_TO_UNICODE[11507] := 16#7127;
   // GBK_TO_UNICODE[11508] := 16#9F75;
   // GBK_TO_UNICODE[11509] := 16#7128;
   // GBK_TO_UNICODE[11510] := 16#9F76;
   // GBK_TO_UNICODE[11511] := 16#7129;
   // GBK_TO_UNICODE[11512] := 16#9F77;
   // GBK_TO_UNICODE[11513] := 16#712A;
   // GBK_TO_UNICODE[11514] := 16#9F78;
   // GBK_TO_UNICODE[11515] := 16#712B;
   // GBK_TO_UNICODE[11516] := 16#9F79;
   // GBK_TO_UNICODE[11517] := 16#712C;
   // GBK_TO_UNICODE[11518] := 16#9F7A;
   // GBK_TO_UNICODE[11519] := 16#712D;
   // GBK_TO_UNICODE[11520] := 16#9F7B;
   // GBK_TO_UNICODE[11521] := 16#712E;
   // GBK_TO_UNICODE[11522] := 16#9F7C;
   // GBK_TO_UNICODE[11523] := 16#7132;
   // GBK_TO_UNICODE[11524] := 16#9F7D;
   // GBK_TO_UNICODE[11525] := 16#7133;
   // GBK_TO_UNICODE[11526] := 16#9F7E;
   // GBK_TO_UNICODE[11527] := 16#7134;
   // GBK_TO_UNICODE[11528] := 16#9F80;
   // GBK_TO_UNICODE[11529] := 16#7135;
   // GBK_TO_UNICODE[11530] := 16#9F81;
   // GBK_TO_UNICODE[11531] := 16#7137;
   // GBK_TO_UNICODE[11532] := 16#9F82;
   // GBK_TO_UNICODE[11533] := 16#7138;
   // GBK_TO_UNICODE[11534] := 16#9F83;
   // GBK_TO_UNICODE[11535] := 16#7139;
   // GBK_TO_UNICODE[11536] := 16#9F84;
   // GBK_TO_UNICODE[11537] := 16#713A;
   // GBK_TO_UNICODE[11538] := 16#9F85;
   // GBK_TO_UNICODE[11539] := 16#713B;
   // GBK_TO_UNICODE[11540] := 16#9F86;
   // GBK_TO_UNICODE[11541] := 16#713C;
   // GBK_TO_UNICODE[11542] := 16#9F87;
   // GBK_TO_UNICODE[11543] := 16#713D;
   // GBK_TO_UNICODE[11544] := 16#9F88;
   // GBK_TO_UNICODE[11545] := 16#713E;
   // GBK_TO_UNICODE[11546] := 16#9F89;
   // GBK_TO_UNICODE[11547] := 16#713F;
   // GBK_TO_UNICODE[11548] := 16#9F8A;
   // GBK_TO_UNICODE[11549] := 16#7140;
   // GBK_TO_UNICODE[11550] := 16#9F8B;
   // GBK_TO_UNICODE[11551] := 16#7141;
   // GBK_TO_UNICODE[11552] := 16#9F8C;
   // GBK_TO_UNICODE[11553] := 16#7142;
   // GBK_TO_UNICODE[11554] := 16#9F8D;
   // GBK_TO_UNICODE[11555] := 16#7143;
   // GBK_TO_UNICODE[11556] := 16#9F8E;
   // GBK_TO_UNICODE[11557] := 16#7144;
   // GBK_TO_UNICODE[11558] := 16#9F8F;
   // GBK_TO_UNICODE[11559] := 16#7146;
   // GBK_TO_UNICODE[11560] := 16#9F90;
   // GBK_TO_UNICODE[11561] := 16#7147;
   // GBK_TO_UNICODE[11562] := 16#9F91;
   // GBK_TO_UNICODE[11563] := 16#7148;
   // GBK_TO_UNICODE[11564] := 16#9F92;
   // GBK_TO_UNICODE[11565] := 16#7149;
   // GBK_TO_UNICODE[11566] := 16#9F93;
   // GBK_TO_UNICODE[11567] := 16#714B;
   // GBK_TO_UNICODE[11568] := 16#9F94;
   // GBK_TO_UNICODE[11569] := 16#714D;
   // GBK_TO_UNICODE[11570] := 16#9F95;
   // GBK_TO_UNICODE[11571] := 16#714F;
   // GBK_TO_UNICODE[11572] := 16#9F96;
   // GBK_TO_UNICODE[11573] := 16#7150;
   // GBK_TO_UNICODE[11574] := 16#9F97;
   // GBK_TO_UNICODE[11575] := 16#7151;
   // GBK_TO_UNICODE[11576] := 16#9F98;
   // GBK_TO_UNICODE[11577] := 16#7152;
   // GBK_TO_UNICODE[11578] := 16#9F99;
   // GBK_TO_UNICODE[11579] := 16#7153;
   // GBK_TO_UNICODE[11580] := 16#9F9A;
   // GBK_TO_UNICODE[11581] := 16#7154;
   // GBK_TO_UNICODE[11582] := 16#9F9B;
   // GBK_TO_UNICODE[11583] := 16#7155;
   // GBK_TO_UNICODE[11584] := 16#9F9C;
   // GBK_TO_UNICODE[11585] := 16#7156;
   // GBK_TO_UNICODE[11586] := 16#9F9D;
   // GBK_TO_UNICODE[11587] := 16#7157;
   // GBK_TO_UNICODE[11588] := 16#9F9E;
   // GBK_TO_UNICODE[11589] := 16#7158;
   // GBK_TO_UNICODE[11590] := 16#9F9F;
   // GBK_TO_UNICODE[11591] := 16#7159;
   // GBK_TO_UNICODE[11592] := 16#9FA0;
   // GBK_TO_UNICODE[11593] := 16#715A;
   // GBK_TO_UNICODE[11594] := 16#9FA1;
   // GBK_TO_UNICODE[11595] := 16#715B;
   // GBK_TO_UNICODE[11596] := 16#9FA2;
   // GBK_TO_UNICODE[11597] := 16#715D;
   // GBK_TO_UNICODE[11598] := 16#9FA3;
   // GBK_TO_UNICODE[11599] := 16#715F;
   // GBK_TO_UNICODE[11600] := 16#9FA4;
   // GBK_TO_UNICODE[11601] := 16#7160;
   // GBK_TO_UNICODE[11602] := 16#9FA5;
   // GBK_TO_UNICODE[11603] := 16#7161;
   // GBK_TO_UNICODE[11604] := 16#9FA6;
   // GBK_TO_UNICODE[11605] := 16#7162;
   // GBK_TO_UNICODE[11606] := 16#9FA7;
   // GBK_TO_UNICODE[11607] := 16#7163;
   // GBK_TO_UNICODE[11608] := 16#9FA8;
   // GBK_TO_UNICODE[11609] := 16#7165;
   // GBK_TO_UNICODE[11610] := 16#9FA9;
   // GBK_TO_UNICODE[11611] := 16#7169;
   // GBK_TO_UNICODE[11612] := 16#9FAA;
   // GBK_TO_UNICODE[11613] := 16#716A;
   // GBK_TO_UNICODE[11614] := 16#9FAB;
   // GBK_TO_UNICODE[11615] := 16#716B;
   // GBK_TO_UNICODE[11616] := 16#9FAC;
   // GBK_TO_UNICODE[11617] := 16#716C;
   // GBK_TO_UNICODE[11618] := 16#9FAD;
   // GBK_TO_UNICODE[11619] := 16#716D;
   // GBK_TO_UNICODE[11620] := 16#9FAE;
   // GBK_TO_UNICODE[11621] := 16#716F;
   // GBK_TO_UNICODE[11622] := 16#9FAF;
   // GBK_TO_UNICODE[11623] := 16#7170;
   // GBK_TO_UNICODE[11624] := 16#9FB0;
   // GBK_TO_UNICODE[11625] := 16#7171;
   // GBK_TO_UNICODE[11626] := 16#9FB1;
   // GBK_TO_UNICODE[11627] := 16#7174;
   // GBK_TO_UNICODE[11628] := 16#9FB2;
   // GBK_TO_UNICODE[11629] := 16#7175;
   // GBK_TO_UNICODE[11630] := 16#9FB3;
   // GBK_TO_UNICODE[11631] := 16#7176;
   // GBK_TO_UNICODE[11632] := 16#9FB4;
   // GBK_TO_UNICODE[11633] := 16#7177;
   // GBK_TO_UNICODE[11634] := 16#9FB5;
   // GBK_TO_UNICODE[11635] := 16#7179;
   // GBK_TO_UNICODE[11636] := 16#9FB6;
   // GBK_TO_UNICODE[11637] := 16#717B;
   // GBK_TO_UNICODE[11638] := 16#9FB7;
   // GBK_TO_UNICODE[11639] := 16#717C;
   // GBK_TO_UNICODE[11640] := 16#9FB8;
   // GBK_TO_UNICODE[11641] := 16#717E;
   // GBK_TO_UNICODE[11642] := 16#9FB9;
   // GBK_TO_UNICODE[11643] := 16#717F;
   // GBK_TO_UNICODE[11644] := 16#9FBA;
   // GBK_TO_UNICODE[11645] := 16#7180;
   // GBK_TO_UNICODE[11646] := 16#9FBB;
   // GBK_TO_UNICODE[11647] := 16#7181;
   // GBK_TO_UNICODE[11648] := 16#9FBC;
   // GBK_TO_UNICODE[11649] := 16#7182;
   // GBK_TO_UNICODE[11650] := 16#9FBD;
   // GBK_TO_UNICODE[11651] := 16#7183;
   // GBK_TO_UNICODE[11652] := 16#9FBE;
   // GBK_TO_UNICODE[11653] := 16#7185;
   // GBK_TO_UNICODE[11654] := 16#9FBF;
   // GBK_TO_UNICODE[11655] := 16#7186;
   // GBK_TO_UNICODE[11656] := 16#9FC0;
   // GBK_TO_UNICODE[11657] := 16#7187;
   // GBK_TO_UNICODE[11658] := 16#9FC1;
   // GBK_TO_UNICODE[11659] := 16#7188;
   // GBK_TO_UNICODE[11660] := 16#9FC2;
   // GBK_TO_UNICODE[11661] := 16#7189;
   // GBK_TO_UNICODE[11662] := 16#9FC3;
   // GBK_TO_UNICODE[11663] := 16#718B;
   // GBK_TO_UNICODE[11664] := 16#9FC4;
   // GBK_TO_UNICODE[11665] := 16#718C;
   // GBK_TO_UNICODE[11666] := 16#9FC5;
   // GBK_TO_UNICODE[11667] := 16#718D;
   // GBK_TO_UNICODE[11668] := 16#9FC6;
   // GBK_TO_UNICODE[11669] := 16#718E;
   // GBK_TO_UNICODE[11670] := 16#9FC7;
   // GBK_TO_UNICODE[11671] := 16#7190;
   // GBK_TO_UNICODE[11672] := 16#9FC8;
   // GBK_TO_UNICODE[11673] := 16#7191;
   // GBK_TO_UNICODE[11674] := 16#9FC9;
   // GBK_TO_UNICODE[11675] := 16#7192;
   // GBK_TO_UNICODE[11676] := 16#9FCA;
   // GBK_TO_UNICODE[11677] := 16#7193;
   // GBK_TO_UNICODE[11678] := 16#9FCB;
   // GBK_TO_UNICODE[11679] := 16#7195;
   // GBK_TO_UNICODE[11680] := 16#9FCC;
   // GBK_TO_UNICODE[11681] := 16#7196;
   // GBK_TO_UNICODE[11682] := 16#9FCD;
   // GBK_TO_UNICODE[11683] := 16#7197;
   // GBK_TO_UNICODE[11684] := 16#9FCE;
   // GBK_TO_UNICODE[11685] := 16#719A;
   // GBK_TO_UNICODE[11686] := 16#9FCF;
   // GBK_TO_UNICODE[11687] := 16#719B;
   // GBK_TO_UNICODE[11688] := 16#9FD0;
   // GBK_TO_UNICODE[11689] := 16#719C;
   // GBK_TO_UNICODE[11690] := 16#9FD1;
   // GBK_TO_UNICODE[11691] := 16#719D;
   // GBK_TO_UNICODE[11692] := 16#9FD2;
   // GBK_TO_UNICODE[11693] := 16#719E;
   // GBK_TO_UNICODE[11694] := 16#9FD3;
   // GBK_TO_UNICODE[11695] := 16#71A1;
   // GBK_TO_UNICODE[11696] := 16#9FD4;
   // GBK_TO_UNICODE[11697] := 16#71A2;
   // GBK_TO_UNICODE[11698] := 16#9FD5;
   // GBK_TO_UNICODE[11699] := 16#71A3;
   // GBK_TO_UNICODE[11700] := 16#9FD6;
   // GBK_TO_UNICODE[11701] := 16#71A4;
   // GBK_TO_UNICODE[11702] := 16#9FD7;
   // GBK_TO_UNICODE[11703] := 16#71A5;
   // GBK_TO_UNICODE[11704] := 16#9FD8;
   // GBK_TO_UNICODE[11705] := 16#71A6;
   // GBK_TO_UNICODE[11706] := 16#9FD9;
   // GBK_TO_UNICODE[11707] := 16#71A7;
   // GBK_TO_UNICODE[11708] := 16#9FDA;
   // GBK_TO_UNICODE[11709] := 16#71A9;
   // GBK_TO_UNICODE[11710] := 16#9FDB;
   // GBK_TO_UNICODE[11711] := 16#71AA;
   // GBK_TO_UNICODE[11712] := 16#9FDC;
   // GBK_TO_UNICODE[11713] := 16#71AB;
   // GBK_TO_UNICODE[11714] := 16#9FDD;
   // GBK_TO_UNICODE[11715] := 16#71AD;
   // GBK_TO_UNICODE[11716] := 16#9FDE;
   // GBK_TO_UNICODE[11717] := 16#71AE;
   // GBK_TO_UNICODE[11718] := 16#9FDF;
   // GBK_TO_UNICODE[11719] := 16#71AF;
   // GBK_TO_UNICODE[11720] := 16#9FE0;
   // GBK_TO_UNICODE[11721] := 16#71B0;
   // GBK_TO_UNICODE[11722] := 16#9FE1;
   // GBK_TO_UNICODE[11723] := 16#71B1;
   // GBK_TO_UNICODE[11724] := 16#9FE2;
   // GBK_TO_UNICODE[11725] := 16#71B2;
   // GBK_TO_UNICODE[11726] := 16#9FE3;
   // GBK_TO_UNICODE[11727] := 16#71B4;
   // GBK_TO_UNICODE[11728] := 16#9FE4;
   // GBK_TO_UNICODE[11729] := 16#71B6;
   // GBK_TO_UNICODE[11730] := 16#9FE5;
   // GBK_TO_UNICODE[11731] := 16#71B7;
   // GBK_TO_UNICODE[11732] := 16#9FE6;
   // GBK_TO_UNICODE[11733] := 16#71B8;
   // GBK_TO_UNICODE[11734] := 16#9FE7;
   // GBK_TO_UNICODE[11735] := 16#71BA;
   // GBK_TO_UNICODE[11736] := 16#9FE8;
   // GBK_TO_UNICODE[11737] := 16#71BB;
   // GBK_TO_UNICODE[11738] := 16#9FE9;
   // GBK_TO_UNICODE[11739] := 16#71BC;
   // GBK_TO_UNICODE[11740] := 16#9FEA;
   // GBK_TO_UNICODE[11741] := 16#71BD;
   // GBK_TO_UNICODE[11742] := 16#9FEB;
   // GBK_TO_UNICODE[11743] := 16#71BE;
   // GBK_TO_UNICODE[11744] := 16#9FEC;
   // GBK_TO_UNICODE[11745] := 16#71BF;
   // GBK_TO_UNICODE[11746] := 16#9FED;
   // GBK_TO_UNICODE[11747] := 16#71C0;
   // GBK_TO_UNICODE[11748] := 16#9FEE;
   // GBK_TO_UNICODE[11749] := 16#71C1;
   // GBK_TO_UNICODE[11750] := 16#9FEF;
   // GBK_TO_UNICODE[11751] := 16#71C2;
   // GBK_TO_UNICODE[11752] := 16#9FF0;
   // GBK_TO_UNICODE[11753] := 16#71C4;
   // GBK_TO_UNICODE[11754] := 16#9FF1;
   // GBK_TO_UNICODE[11755] := 16#71C5;
   // GBK_TO_UNICODE[11756] := 16#9FF2;
   // GBK_TO_UNICODE[11757] := 16#71C6;
   // GBK_TO_UNICODE[11758] := 16#9FF3;
   // GBK_TO_UNICODE[11759] := 16#71C7;
   // GBK_TO_UNICODE[11760] := 16#9FF4;
   // GBK_TO_UNICODE[11761] := 16#71C8;
   // GBK_TO_UNICODE[11762] := 16#9FF5;
   // GBK_TO_UNICODE[11763] := 16#71C9;
   // GBK_TO_UNICODE[11764] := 16#9FF6;
   // GBK_TO_UNICODE[11765] := 16#71CA;
   // GBK_TO_UNICODE[11766] := 16#9FF7;
   // GBK_TO_UNICODE[11767] := 16#71CB;
   // GBK_TO_UNICODE[11768] := 16#9FF8;
   // GBK_TO_UNICODE[11769] := 16#71CC;
   // GBK_TO_UNICODE[11770] := 16#9FF9;
   // GBK_TO_UNICODE[11771] := 16#71CD;
   // GBK_TO_UNICODE[11772] := 16#9FFA;
   // GBK_TO_UNICODE[11773] := 16#71CF;
   // GBK_TO_UNICODE[11774] := 16#9FFB;
   // GBK_TO_UNICODE[11775] := 16#71D0;
   // GBK_TO_UNICODE[11776] := 16#9FFC;
   // GBK_TO_UNICODE[11777] := 16#71D1;
   // GBK_TO_UNICODE[11778] := 16#9FFD;
   // GBK_TO_UNICODE[11779] := 16#71D2;
   // GBK_TO_UNICODE[11780] := 16#9FFE;
   // GBK_TO_UNICODE[11781] := 16#71D3;
   // GBK_TO_UNICODE[11782] := 16#A040;
   // GBK_TO_UNICODE[11783] := 16#71D6;
   // GBK_TO_UNICODE[11784] := 16#A041;
   // GBK_TO_UNICODE[11785] := 16#71D7;
   // GBK_TO_UNICODE[11786] := 16#A042;
   // GBK_TO_UNICODE[11787] := 16#71D8;
   // GBK_TO_UNICODE[11788] := 16#A043;
   // GBK_TO_UNICODE[11789] := 16#71D9;
   // GBK_TO_UNICODE[11790] := 16#A044;
   // GBK_TO_UNICODE[11791] := 16#71DA;
   // GBK_TO_UNICODE[11792] := 16#A045;
   // GBK_TO_UNICODE[11793] := 16#71DB;
   // GBK_TO_UNICODE[11794] := 16#A046;
   // GBK_TO_UNICODE[11795] := 16#71DC;
   // GBK_TO_UNICODE[11796] := 16#A047;
   // GBK_TO_UNICODE[11797] := 16#71DD;
   // GBK_TO_UNICODE[11798] := 16#A048;
   // GBK_TO_UNICODE[11799] := 16#71DE;
   // GBK_TO_UNICODE[11800] := 16#A049;
   // GBK_TO_UNICODE[11801] := 16#71DF;
   // GBK_TO_UNICODE[11802] := 16#A04A;
   // GBK_TO_UNICODE[11803] := 16#71E1;
   // GBK_TO_UNICODE[11804] := 16#A04B;
   // GBK_TO_UNICODE[11805] := 16#71E2;
   // GBK_TO_UNICODE[11806] := 16#A04C;
   // GBK_TO_UNICODE[11807] := 16#71E3;
   // GBK_TO_UNICODE[11808] := 16#A04D;
   // GBK_TO_UNICODE[11809] := 16#71E4;
   // GBK_TO_UNICODE[11810] := 16#A04E;
   // GBK_TO_UNICODE[11811] := 16#71E6;
   // GBK_TO_UNICODE[11812] := 16#A04F;
   // GBK_TO_UNICODE[11813] := 16#71E8;
   // GBK_TO_UNICODE[11814] := 16#A050;
   // GBK_TO_UNICODE[11815] := 16#71E9;
   // GBK_TO_UNICODE[11816] := 16#A051;
   // GBK_TO_UNICODE[11817] := 16#71EA;
   // GBK_TO_UNICODE[11818] := 16#A052;
   // GBK_TO_UNICODE[11819] := 16#71EB;
   // GBK_TO_UNICODE[11820] := 16#A053;
   // GBK_TO_UNICODE[11821] := 16#71EC;
   // GBK_TO_UNICODE[11822] := 16#A054;
   // GBK_TO_UNICODE[11823] := 16#71ED;
   // GBK_TO_UNICODE[11824] := 16#A055;
   // GBK_TO_UNICODE[11825] := 16#71EF;
   // GBK_TO_UNICODE[11826] := 16#A056;
   // GBK_TO_UNICODE[11827] := 16#71F0;
   // GBK_TO_UNICODE[11828] := 16#A057;
   // GBK_TO_UNICODE[11829] := 16#71F1;
   // GBK_TO_UNICODE[11830] := 16#A058;
   // GBK_TO_UNICODE[11831] := 16#71F2;
   // GBK_TO_UNICODE[11832] := 16#A059;
   // GBK_TO_UNICODE[11833] := 16#71F3;
   // GBK_TO_UNICODE[11834] := 16#A05A;
   // GBK_TO_UNICODE[11835] := 16#71F4;
   // GBK_TO_UNICODE[11836] := 16#A05B;
   // GBK_TO_UNICODE[11837] := 16#71F5;
   // GBK_TO_UNICODE[11838] := 16#A05C;
   // GBK_TO_UNICODE[11839] := 16#71F6;
   // GBK_TO_UNICODE[11840] := 16#A05D;
   // GBK_TO_UNICODE[11841] := 16#71F7;
   // GBK_TO_UNICODE[11842] := 16#A05E;
   // GBK_TO_UNICODE[11843] := 16#71F8;
   // GBK_TO_UNICODE[11844] := 16#A05F;
   // GBK_TO_UNICODE[11845] := 16#71FA;
   // GBK_TO_UNICODE[11846] := 16#A060;
   // GBK_TO_UNICODE[11847] := 16#71FB;
   // GBK_TO_UNICODE[11848] := 16#A061;
   // GBK_TO_UNICODE[11849] := 16#71FC;
   // GBK_TO_UNICODE[11850] := 16#A062;
   // GBK_TO_UNICODE[11851] := 16#71FD;
   // GBK_TO_UNICODE[11852] := 16#A063;
   // GBK_TO_UNICODE[11853] := 16#71FE;
   // GBK_TO_UNICODE[11854] := 16#A064;
   // GBK_TO_UNICODE[11855] := 16#71FF;
   // GBK_TO_UNICODE[11856] := 16#A065;
   // GBK_TO_UNICODE[11857] := 16#7200;
   // GBK_TO_UNICODE[11858] := 16#A066;
   // GBK_TO_UNICODE[11859] := 16#7201;
   // GBK_TO_UNICODE[11860] := 16#A067;
   // GBK_TO_UNICODE[11861] := 16#7202;
   // GBK_TO_UNICODE[11862] := 16#A068;
   // GBK_TO_UNICODE[11863] := 16#7203;
   // GBK_TO_UNICODE[11864] := 16#A069;
   // GBK_TO_UNICODE[11865] := 16#7204;
   // GBK_TO_UNICODE[11866] := 16#A06A;
   // GBK_TO_UNICODE[11867] := 16#7205;
   // GBK_TO_UNICODE[11868] := 16#A06B;
   // GBK_TO_UNICODE[11869] := 16#7207;
   // GBK_TO_UNICODE[11870] := 16#A06C;
   // GBK_TO_UNICODE[11871] := 16#7208;
   // GBK_TO_UNICODE[11872] := 16#A06D;
   // GBK_TO_UNICODE[11873] := 16#7209;
   // GBK_TO_UNICODE[11874] := 16#A06E;
   // GBK_TO_UNICODE[11875] := 16#720A;
   // GBK_TO_UNICODE[11876] := 16#A06F;
   // GBK_TO_UNICODE[11877] := 16#720B;
   // GBK_TO_UNICODE[11878] := 16#A070;
   // GBK_TO_UNICODE[11879] := 16#720C;
   // GBK_TO_UNICODE[11880] := 16#A071;
   // GBK_TO_UNICODE[11881] := 16#720D;
   // GBK_TO_UNICODE[11882] := 16#A072;
   // GBK_TO_UNICODE[11883] := 16#720E;
   // GBK_TO_UNICODE[11884] := 16#A073;
   // GBK_TO_UNICODE[11885] := 16#720F;
   // GBK_TO_UNICODE[11886] := 16#A074;
   // GBK_TO_UNICODE[11887] := 16#7210;
   // GBK_TO_UNICODE[11888] := 16#A075;
   // GBK_TO_UNICODE[11889] := 16#7211;
   // GBK_TO_UNICODE[11890] := 16#A076;
   // GBK_TO_UNICODE[11891] := 16#7212;
   // GBK_TO_UNICODE[11892] := 16#A077;
   // GBK_TO_UNICODE[11893] := 16#7213;
   // GBK_TO_UNICODE[11894] := 16#A078;
   // GBK_TO_UNICODE[11895] := 16#7214;
   // GBK_TO_UNICODE[11896] := 16#A079;
   // GBK_TO_UNICODE[11897] := 16#7215;
   // GBK_TO_UNICODE[11898] := 16#A07A;
   // GBK_TO_UNICODE[11899] := 16#7216;
   // GBK_TO_UNICODE[11900] := 16#A07B;
   // GBK_TO_UNICODE[11901] := 16#7217;
   // GBK_TO_UNICODE[11902] := 16#A07C;
   // GBK_TO_UNICODE[11903] := 16#7218;
   // GBK_TO_UNICODE[11904] := 16#A07D;
   // GBK_TO_UNICODE[11905] := 16#7219;
   // GBK_TO_UNICODE[11906] := 16#A07E;
   // GBK_TO_UNICODE[11907] := 16#721A;
   // GBK_TO_UNICODE[11908] := 16#A080;
   // GBK_TO_UNICODE[11909] := 16#721B;
   // GBK_TO_UNICODE[11910] := 16#A081;
   // GBK_TO_UNICODE[11911] := 16#721C;
   // GBK_TO_UNICODE[11912] := 16#A082;
   // GBK_TO_UNICODE[11913] := 16#721E;
   // GBK_TO_UNICODE[11914] := 16#A083;
   // GBK_TO_UNICODE[11915] := 16#721F;
   // GBK_TO_UNICODE[11916] := 16#A084;
   // GBK_TO_UNICODE[11917] := 16#7220;
   // GBK_TO_UNICODE[11918] := 16#A085;
   // GBK_TO_UNICODE[11919] := 16#7221;
   // GBK_TO_UNICODE[11920] := 16#A086;
   // GBK_TO_UNICODE[11921] := 16#7222;
   // GBK_TO_UNICODE[11922] := 16#A087;
   // GBK_TO_UNICODE[11923] := 16#7223;
   // GBK_TO_UNICODE[11924] := 16#A088;
   // GBK_TO_UNICODE[11925] := 16#7224;
   // GBK_TO_UNICODE[11926] := 16#A089;
   // GBK_TO_UNICODE[11927] := 16#7225;
   // GBK_TO_UNICODE[11928] := 16#A08A;
   // GBK_TO_UNICODE[11929] := 16#7226;
   // GBK_TO_UNICODE[11930] := 16#A08B;
   // GBK_TO_UNICODE[11931] := 16#7227;
   // GBK_TO_UNICODE[11932] := 16#A08C;
   // GBK_TO_UNICODE[11933] := 16#7229;
   // GBK_TO_UNICODE[11934] := 16#A08D;
   // GBK_TO_UNICODE[11935] := 16#722B;
   // GBK_TO_UNICODE[11936] := 16#A08E;
   // GBK_TO_UNICODE[11937] := 16#722D;
   // GBK_TO_UNICODE[11938] := 16#A08F;
   // GBK_TO_UNICODE[11939] := 16#722E;
   // GBK_TO_UNICODE[11940] := 16#A090;
   // GBK_TO_UNICODE[11941] := 16#722F;
   // GBK_TO_UNICODE[11942] := 16#A091;
   // GBK_TO_UNICODE[11943] := 16#7232;
   // GBK_TO_UNICODE[11944] := 16#A092;
   // GBK_TO_UNICODE[11945] := 16#7233;
   // GBK_TO_UNICODE[11946] := 16#A093;
   // GBK_TO_UNICODE[11947] := 16#7234;
   // GBK_TO_UNICODE[11948] := 16#A094;
   // GBK_TO_UNICODE[11949] := 16#723A;
   // GBK_TO_UNICODE[11950] := 16#A095;
   // GBK_TO_UNICODE[11951] := 16#723C;
   // GBK_TO_UNICODE[11952] := 16#A096;
   // GBK_TO_UNICODE[11953] := 16#723E;
   // GBK_TO_UNICODE[11954] := 16#A097;
   // GBK_TO_UNICODE[11955] := 16#7240;
   // GBK_TO_UNICODE[11956] := 16#A098;
   // GBK_TO_UNICODE[11957] := 16#7241;
   // GBK_TO_UNICODE[11958] := 16#A099;
   // GBK_TO_UNICODE[11959] := 16#7242;
   // GBK_TO_UNICODE[11960] := 16#A09A;
   // GBK_TO_UNICODE[11961] := 16#7243;
   // GBK_TO_UNICODE[11962] := 16#A09B;
   // GBK_TO_UNICODE[11963] := 16#7244;
   // GBK_TO_UNICODE[11964] := 16#A09C;
   // GBK_TO_UNICODE[11965] := 16#7245;
   // GBK_TO_UNICODE[11966] := 16#A09D;
   // GBK_TO_UNICODE[11967] := 16#7246;
   // GBK_TO_UNICODE[11968] := 16#A09E;
   // GBK_TO_UNICODE[11969] := 16#7249;
   // GBK_TO_UNICODE[11970] := 16#A09F;
   // GBK_TO_UNICODE[11971] := 16#724A;
   // GBK_TO_UNICODE[11972] := 16#A0A0;
   // GBK_TO_UNICODE[11973] := 16#724B;
   // GBK_TO_UNICODE[11974] := 16#A0A1;
   // GBK_TO_UNICODE[11975] := 16#724E;
   // GBK_TO_UNICODE[11976] := 16#A0A2;
   // GBK_TO_UNICODE[11977] := 16#724F;
   // GBK_TO_UNICODE[11978] := 16#A0A3;
   // GBK_TO_UNICODE[11979] := 16#7250;
   // GBK_TO_UNICODE[11980] := 16#A0A4;
   // GBK_TO_UNICODE[11981] := 16#7251;
   // GBK_TO_UNICODE[11982] := 16#A0A5;
   // GBK_TO_UNICODE[11983] := 16#7253;
   // GBK_TO_UNICODE[11984] := 16#A0A6;
   // GBK_TO_UNICODE[11985] := 16#7254;
   // GBK_TO_UNICODE[11986] := 16#A0A7;
   // GBK_TO_UNICODE[11987] := 16#7255;
   // GBK_TO_UNICODE[11988] := 16#A0A8;
   // GBK_TO_UNICODE[11989] := 16#7257;
   // GBK_TO_UNICODE[11990] := 16#A0A9;
   // GBK_TO_UNICODE[11991] := 16#7258;
   // GBK_TO_UNICODE[11992] := 16#A0AA;
   // GBK_TO_UNICODE[11993] := 16#725A;
   // GBK_TO_UNICODE[11994] := 16#A0AB;
   // GBK_TO_UNICODE[11995] := 16#725C;
   // GBK_TO_UNICODE[11996] := 16#A0AC;
   // GBK_TO_UNICODE[11997] := 16#725E;
   // GBK_TO_UNICODE[11998] := 16#A0AD;
   // GBK_TO_UNICODE[11999] := 16#7260;
   // GBK_TO_UNICODE[12000] := 16#A0AE;
   // GBK_TO_UNICODE[12001] := 16#7263;
   // GBK_TO_UNICODE[12002] := 16#A0AF;
   // GBK_TO_UNICODE[12003] := 16#7264;
   // GBK_TO_UNICODE[12004] := 16#A0B0;
   // GBK_TO_UNICODE[12005] := 16#7265;
   // GBK_TO_UNICODE[12006] := 16#A0B1;
   // GBK_TO_UNICODE[12007] := 16#7268;
   // GBK_TO_UNICODE[12008] := 16#A0B2;
   // GBK_TO_UNICODE[12009] := 16#726A;
   // GBK_TO_UNICODE[12010] := 16#A0B3;
   // GBK_TO_UNICODE[12011] := 16#726B;
   // GBK_TO_UNICODE[12012] := 16#A0B4;
   // GBK_TO_UNICODE[12013] := 16#726C;
   // GBK_TO_UNICODE[12014] := 16#A0B5;
   // GBK_TO_UNICODE[12015] := 16#726D;
   // GBK_TO_UNICODE[12016] := 16#A0B6;
   // GBK_TO_UNICODE[12017] := 16#7270;
   // GBK_TO_UNICODE[12018] := 16#A0B7;
   // GBK_TO_UNICODE[12019] := 16#7271;
   // GBK_TO_UNICODE[12020] := 16#A0B8;
   // GBK_TO_UNICODE[12021] := 16#7273;
   // GBK_TO_UNICODE[12022] := 16#A0B9;
   // GBK_TO_UNICODE[12023] := 16#7274;
   // GBK_TO_UNICODE[12024] := 16#A0BA;
   // GBK_TO_UNICODE[12025] := 16#7276;
   // GBK_TO_UNICODE[12026] := 16#A0BB;
   // GBK_TO_UNICODE[12027] := 16#7277;
   // GBK_TO_UNICODE[12028] := 16#A0BC;
   // GBK_TO_UNICODE[12029] := 16#7278;
   // GBK_TO_UNICODE[12030] := 16#A0BD;
   // GBK_TO_UNICODE[12031] := 16#727B;
   // GBK_TO_UNICODE[12032] := 16#A0BE;
   // GBK_TO_UNICODE[12033] := 16#727C;
   // GBK_TO_UNICODE[12034] := 16#A0BF;
   // GBK_TO_UNICODE[12035] := 16#727D;
   // GBK_TO_UNICODE[12036] := 16#A0C0;
   // GBK_TO_UNICODE[12037] := 16#7282;
   // GBK_TO_UNICODE[12038] := 16#A0C1;
   // GBK_TO_UNICODE[12039] := 16#7283;
   // GBK_TO_UNICODE[12040] := 16#A0C2;
   // GBK_TO_UNICODE[12041] := 16#7285;
   // GBK_TO_UNICODE[12042] := 16#A0C3;
   // GBK_TO_UNICODE[12043] := 16#7286;
   // GBK_TO_UNICODE[12044] := 16#A0C4;
   // GBK_TO_UNICODE[12045] := 16#7287;
   // GBK_TO_UNICODE[12046] := 16#A0C5;
   // GBK_TO_UNICODE[12047] := 16#7288;
   // GBK_TO_UNICODE[12048] := 16#A0C6;
   // GBK_TO_UNICODE[12049] := 16#7289;
   // GBK_TO_UNICODE[12050] := 16#A0C7;
   // GBK_TO_UNICODE[12051] := 16#728C;
   // GBK_TO_UNICODE[12052] := 16#A0C8;
   // GBK_TO_UNICODE[12053] := 16#728E;
   // GBK_TO_UNICODE[12054] := 16#A0C9;
   // GBK_TO_UNICODE[12055] := 16#7290;
   // GBK_TO_UNICODE[12056] := 16#A0CA;
   // GBK_TO_UNICODE[12057] := 16#7291;
   // GBK_TO_UNICODE[12058] := 16#A0CB;
   // GBK_TO_UNICODE[12059] := 16#7293;
   // GBK_TO_UNICODE[12060] := 16#A0CC;
   // GBK_TO_UNICODE[12061] := 16#7294;
   // GBK_TO_UNICODE[12062] := 16#A0CD;
   // GBK_TO_UNICODE[12063] := 16#7295;
   // GBK_TO_UNICODE[12064] := 16#A0CE;
   // GBK_TO_UNICODE[12065] := 16#7296;
   // GBK_TO_UNICODE[12066] := 16#A0CF;
   // GBK_TO_UNICODE[12067] := 16#7297;
